LIN {X 0,Y 481.295,Z 335.256,A -85,B 0,C 180,E1 -6793.339,E2 -6793.339} C_VEL
LIN {X 0,Y 481.494,Z 329.441,A -85,B 0,C 180,E1 -6794.339,E2 -6794.339} C_VEL
LIN {X 0,Y 481.671,Z 324.523,A -85,B 0,C 180,E1 -6795.045,E2 -6795.045} C_VEL
LIN {X 0,Y 481.939,Z 317.288,A -85,B 0,C 180,E1 -6795.906,E2 -6795.906} C_VEL
LIN {X 0,Y 482.147,Z 309.914,A -85,B 0,C 180,E1 -6796.628,E2 -6796.628} C_VEL
LIN {X 0,Y 482.417,Z 301.623,A -85,B 0,C 180,E1 -6797.289,E2 -6797.289} C_VEL
LIN {X 0,Y 482.717,Z 290.959,A -85,B 0,C 180,E1 -6797.954,E2 -6797.954} C_VEL
LIN {X 0,Y 482.784,Z 280.373,A -85,B 0,C 180,E1 -6798.426,E2 -6798.426} C_VEL
LIN {X 0,Y 481.052,Z 270.815,A -85,B 0,C 180,E1 -6798.793,E2 -6798.793} C_VEL
LIN {X 0,Y 481.125,Z 264.772,A -85,B 0,C 180,E1 -6801.617,E2 -6801.617} C_VEL
LIN {X 0,Y 481.175,Z 257.779,A -85,B 0,C 180,E1 -6804.879,E2 -6804.879} C_VEL
LIN {X 0,Y 481.271,Z 252.542,A -85,B 0,C 180,E1 -6807.295,E2 -6807.295} C_VEL
LIN {X 0,Y 481.297,Z 246.12,A -85,B 0,C 180,E1 -6810.233,E2 -6810.233} C_VEL
LIN {X 0,Y 481.291,Z 239.614,A -85,B 0,C 180,E1 -6813.084,E2 -6813.084} C_VEL
LIN {X 0,Y 481.364,Z 233.224,A -85,B 0,C 180,E1 -6815.87,E2 -6815.87} C_VEL
LIN {X 0,Y 481.43,Z 228.524,A -85,B 0,C 180,E1 -6817.92,E2 -6817.92} C_VEL
LIN {X 0,Y 481.692,Z 228.485,A -85,B 0,C 180,E1 -6820.392,E2 -6820.392} C_VEL
LIN {X 0,Y 481.681,Z 228.487,A -85,B 0,C 180,E1 -6823.033,E2 -6823.033} C_VEL
LIN {X 0,Y 481.691,Z 228.486,A -85,B 0,C 180,E1 -6825.639,E2 -6825.639} C_VEL
LIN {X 0,Y 481.754,Z 228.48,A -85,B 0,C 180,E1 -6828.215,E2 -6828.215} C_VEL
LIN {X 0,Y 481.766,Z 228.477,A -85,B 0,C 180,E1 -6831.612,E2 -6831.612} C_VEL
LIN {X 0,Y 481.778,Z 228.474,A -85,B 0,C 180,E1 -6834.979,E2 -6834.979} C_VEL
LIN {X 0,Y 481.931,Z 228.456,A -85,B 0,C 180,E1 -6837.492,E2 -6837.492} C_VEL
LIN {X 0,Y 481.889,Z 228.46,A -85,B 0,C 180,E1 -6840.836,E2 -6840.836} C_VEL
LIN {X 0,Y 481.931,Z 228.458,A -85,B 0,C 180,E1 -6842.507,E2 -6842.507} C_VEL
LIN {X 0,Y 481.8,Z 228.472,A -85,B 0,C 180,E1 -6845.861,E2 -6845.861} C_VEL
LIN {X 0,Y 481.765,Z 228.477,A -85,B 0,C 180,E1 -6848.388,E2 -6848.388} C_VEL
LIN {X 0,Y 481.754,Z 228.477,A -85,B 0,C 180,E1 -6851.785,E2 -6851.785} C_VEL
LIN {X 0,Y 481.746,Z 228.478,A -85,B 0,C 180,E1 -6855.224,E2 -6855.224} C_VEL
LIN {X 0,Y 481.711,Z 228.481,A -85,B 0,C 180,E1 -6858.722,E2 -6858.722} C_VEL
LIN {X 0,Y 481.648,Z 228.491,A -85,B 0,C 180,E1 -6861.395,E2 -6861.395} C_VEL
LIN {X 0,Y 481.654,Z 228.489,A -85,B 0,C 180,E1 -6864.114,E2 -6864.114} C_VEL
LIN {X 0,Y 481.718,Z 228.48,A -85,B 0,C 180,E1 -6867.132,E2 -6867.132} C_VEL
LIN {X 0,Y 481.68,Z 228.486,A -85,B 0,C 180,E1 -6869.741,E2 -6869.741} C_VEL
LIN {X 0,Y 481.672,Z 228.486,A -85,B 0,C 180,E1 -6872.674,E2 -6872.674} C_VEL
LIN {X 0,Y 481.638,Z 228.492,A -85,B 0,C 180,E1 -6875.71,E2 -6875.71} C_VEL
LIN {X 0,Y 481.673,Z 228.486,A -85,B 0,C 180,E1 -6878.859,E2 -6878.859} C_VEL
LIN {X 0,Y 481.654,Z 228.49,A -85,B 0,C 180,E1 -6881.913,E2 -6881.913} C_VEL
LIN {X 0,Y 481.656,Z 228.49,A -85,B 0,C 180,E1 -6884.458,E2 -6884.458} C_VEL
LIN {X 0,Y 481.649,Z 228.491,A -85,B 0,C 180,E1 -6887.839,E2 -6887.839} C_VEL
LIN {X 0,Y 481.737,Z 228.644,A -85,B 0,C 180,E1 -6890.145,E2 -6890.145} C_VEL
LIN {X 0,Y 483.016,Z 236.207,A -85,B 0,C 180,E1 -6893.376,E2 -6893.376} C_VEL
LIN {X 0,Y 483.177,Z 240.208,A -85,B 0,C 180,E1 -6894.988,E2 -6894.988} C_VEL
LIN {X 0,Y 482.787,Z 248.025,A -85,B 0,C 180,E1 -6897.992,E2 -6897.992} C_VEL
LIN {X 0,Y 482.344,Z 256.819,A -85,B 0,C 180,E1 -6901.261,E2 -6901.261} C_VEL
LIN {X 0,Y 481.939,Z 266.411,A -85,B 0,C 180,E1 -6904.707,E2 -6904.707} C_VEL
LIN {X 0,Y 481.657,Z 274.969,A -85,B 0,C 180,E1 -6907.705,E2 -6907.705} C_VEL
LIN {X 0,Y 481.398,Z 284.073,A -85,B 0,C 180,E1 -6910.823,E2 -6910.823} C_VEL
LIN {X 0,Y 481.24,Z 293.194,A -85,B 0,C 180,E1 -6913.89,E2 -6913.89} C_VEL
LIN {X 0,Y 481.156,Z 296.798,A -85,B 0,C 180,E1 -6915.082,E2 -6915.082} C_VEL
LIN {X 0,Y 483.171,Z 311.724,A -85,B 0,C 180,E1 -6915.563,E2 -6915.563} C_VEL
LIN {X 0,Y 483.633,Z 316.455,A -85,B 0,C 180,E1 -6915.751,E2 -6915.751} C_VEL
LIN {X 0,Y 483.234,Z 328.917,A -85,B 0,C 180,E1 -6916.33,E2 -6916.33} C_VEL
LIN {X 0,Y 482.765,Z 340.987,A -85,B 0,C 180,E1 -6917.067,E2 -6917.067} C_VEL
LIN {X 0,Y 482.282,Z 352.197,A -85,B 0,C 180,E1 -6917.938,E2 -6917.938} C_VEL
LIN {X 0,Y 481.972,Z 361.764,A -85,B 0,C 180,E1 -6918.86,E2 -6918.86} C_VEL
LIN {X 0,Y 481.571,Z 370.781,A -85,B 0,C 180,E1 -6919.914,E2 -6919.914} C_VEL
LIN {X 0,Y 481.279,Z 379.611,A -85,B 0,C 180,E1 -6921.18,E2 -6921.18} C_VEL
LIN {X 0,Y 481.101,Z 386.663,A -85,B 0,C 180,E1 -6922.445,E2 -6922.445} C_VEL
LIN {X 0,Y 480.921,Z 392.764,A -85,B 0,C 180,E1 -6923.827,E2 -6923.827} C_VEL
LIN {X 0,Y 480.902,Z 396.727,A -85,B 0,C 180,E1 -6924.97,E2 -6924.97} C_VEL
LIN {X 0,Y 480.849,Z 399.059,A -85,B 0,C 180,E1 -6925.809,E2 -6925.809} C_VEL
LIN {X 0,Y 480.894,Z 400.958,A -85,B 0,C 180,E1 -6926.649,E2 -6926.649} C_VEL
LIN {X 0,Y 480.869,Z 402.379,A -85,B 0,C 180,E1 -6927.487,E2 -6927.487} C_VEL
LIN {X 0,Y 480.824,Z 403.378,A -85,B 0,C 180,E1 -6928.325,E2 -6928.325} C_VEL
LIN {X 0,Y 480.763,Z 403.977,A -85,B 0,C 180,E1 -6929.163,E2 -6929.163} C_VEL
LIN {X 0,Y 480.752,Z 404.178,A -85,B 0,C 180,E1 -6930,E2 -6930} C_VEL
LIN {X 0,Y 480.764,Z 403.933,A -85,B 0,C 180,E1 -6930.838,E2 -6930.838} C_VEL
LIN {X 0,Y 480.824,Z 403.286,A -85,B 0,C 180,E1 -6931.675,E2 -6931.675} C_VEL
LIN {X 0,Y 480.869,Z 402.238,A -85,B 0,C 180,E1 -6932.513,E2 -6932.513} C_VEL
LIN {X 0,Y 480.896,Z 400.77,A -85,B 0,C 180,E1 -6933.351,E2 -6933.351} C_VEL
LIN {X 0,Y 480.847,Z 397.7,A -85,B 0,C 180,E1 -6934.611,E2 -6934.611} C_VEL
LIN {X 0,Y 480.931,Z 393.56,A -85,B 0,C 180,E1 -6935.871,E2 -6935.871} C_VEL
LIN {X 0,Y 481.106,Z 387.196,A -85,B 0,C 180,E1 -6937.344,E2 -6937.344} C_VEL
LIN {X 0,Y 481.256,Z 380.258,A -85,B 0,C 180,E1 -6938.609,E2 -6938.609} C_VEL
LIN {X 0,Y 481.508,Z 371.668,A -85,B 0,C 180,E1 -6939.875,E2 -6939.875} C_VEL
LIN {X 0,Y 481.844,Z 362.847,A -85,B 0,C 180,E1 -6940.93,E2 -6940.93} C_VEL
LIN {X 0,Y 482.173,Z 352.482,A -85,B 0,C 180,E1 -6941.948,E2 -6941.948} C_VEL
LIN {X 0,Y 482.589,Z 341.383,A -85,B 0,C 180,E1 -6942.832,E2 -6942.832} C_VEL
LIN {X 0,Y 483.067,Z 329.672,A -85,B 0,C 180,E1 -6943.568,E2 -6943.568} C_VEL
LIN {X 0,Y 483.567,Z 316.581,A -85,B 0,C 180,E1 -6944.197,E2 -6944.197} C_VEL
LIN {X 0,Y 482.164,Z 303.16,A -85,B 0,C 180,E1 -6944.711,E2 -6944.711} C_VEL
LIN {X 0,Y 481.08,Z 295.296,A -85,B 0,C 180,E1 -6944.948,E2 -6944.948} C_VEL
LIN {X 0,Y 481.261,Z 284.885,A -85,B 0,C 180,E1 -6948.338,E2 -6948.338} C_VEL
LIN {X 0,Y 481.46,Z 275.744,A -85,B 0,C 180,E1 -6951.404,E2 -6951.404} C_VEL
LIN {X 0,Y 481.668,Z 266.683,A -85,B 0,C 180,E1 -6954.573,E2 -6954.573} C_VEL
LIN {X 0,Y 481.949,Z 259.603,A -85,B 0,C 180,E1 -6957.186,E2 -6957.186} C_VEL
LIN {X 0,Y 482.36,Z 252.034,A -85,B 0,C 180,E1 -6960.177,E2 -6960.177} C_VEL
LIN {X 0,Y 482.964,Z 245.384,A -85,B 0,C 180,E1 -6963.072,E2 -6963.072} C_VEL
LIN {X 0,Y 483.35,Z 240.369,A -85,B 0,C 180,E1 -6965.564,E2 -6965.564} C_VEL
LIN {X 0,Y 483.107,Z 236.847,A -85,B 0,C 180,E1 -6967.662,E2 -6967.662} C_VEL
LIN {X 0,Y 482.648,Z 233.878,A -85,B 0,C 180,E1 -6969.844,E2 -6969.844} C_VEL
LIN {X 0,Y 482.207,Z 231.543,A -85,B 0,C 180,E1 -6972.101,E2 -6972.101} C_VEL
LIN {X 0,Y 481.93,Z 229.935,A -85,B 0,C 180,E1 -6974.426,E2 -6974.426} C_VEL
LIN {X 0,Y 481.743,Z 229.06,A -85,B 0,C 180,E1 -6976.84,E2 -6976.84} C_VEL
LIN {X 0,Y 481.749,Z 228.914,A -85,B 0,C 180,E1 -6979.342,E2 -6979.342} C_VEL
LIN {X 0,Y 481.838,Z 229.553,A -85,B 0,C 180,E1 -6982.222,E2 -6982.222} C_VEL
LIN {X 0,Y 481.94,Z 230.974,A -85,B 0,C 180,E1 -6985.339,E2 -6985.339} C_VEL
LIN {X 0,Y 481.767,Z 232.856,A -85,B 0,C 180,E1 -6988.32,E2 -6988.32} C_VEL
LIN {X 0,Y 481.589,Z 234.985,A -85,B 0,C 180,E1 -6991.211,E2 -6991.211} C_VEL
LIN {X 0,Y 481.467,Z 237.269,A -85,B 0,C 180,E1 -6994.029,E2 -6994.029} C_VEL
LIN {X 0,Y 481.344,Z 239.756,A -85,B 0,C 180,E1 -6996.905,E2 -6996.905} C_VEL
LIN {X 0,Y 481.253,Z 242.102,A -85,B 0,C 180,E1 -6999.483,E2 -6999.483} C_VEL
LIN {X 0,Y 481.221,Z 244.619,A -85,B 0,C 180,E1 -7002.14,E2 -7002.14} C_VEL
LIN {X 0,Y 481.172,Z 247.192,A -85,B 0,C 180,E1 -7004.757,E2 -7004.757} C_VEL
LIN {X 0,Y 481.113,Z 248.8,A -85,B 0,C 180,E1 -7006.201,E2 -7006.201} C_VEL
LIN {X 0,Y 484.037,Z 261.107,A -85,B 0,C 180,E1 -7006.7,E2 -7006.7} C_VEL
LIN {X 0,Y 483.743,Z 273.649,A -85,B 0,C 180,E1 -7007.254,E2 -7007.254} C_VEL
LIN {X 0,Y 483.415,Z 285.282,A -85,B 0,C 180,E1 -7007.937,E2 -7007.937} C_VEL
LIN {X 0,Y 482.913,Z 296.516,A -85,B 0,C 180,E1 -7008.776,E2 -7008.776} C_VEL
LIN {X 0,Y 482.478,Z 306.707,A -85,B 0,C 180,E1 -7009.721,E2 -7009.721} C_VEL
LIN {X 0,Y 482.162,Z 315.925,A -85,B 0,C 180,E1 -7010.774,E2 -7010.774} C_VEL
LIN {X 0,Y 481.71,Z 324.854,A -85,B 0,C 180,E1 -7012.033,E2 -7012.033} C_VEL
LIN {X 0,Y 481.487,Z 332.04,A -85,B 0,C 180,E1 -7013.294,E2 -7013.294} C_VEL
LIN {X 0,Y 481.262,Z 337.788,A -85,B 0,C 180,E1 -7014.553,E2 -7014.553} C_VEL
LIN {X 0,Y 481.111,Z 342.296,A -85,B 0,C 180,E1 -7015.812,E2 -7015.812} C_VEL
LIN {X 0,Y 481.138,Z 344.659,A -85,B 0,C 180,E1 -7016.65,E2 -7016.65} C_VEL
LIN {X 0,Y 480.969,Z 346.601,A -85,B 0,C 180,E1 -7017.488,E2 -7017.488} C_VEL
LIN {X 0,Y 480.838,Z 348.127,A -85,B 0,C 180,E1 -7018.325,E2 -7018.325} C_VEL
LIN {X 0,Y 480.778,Z 349.206,A -85,B 0,C 180,E1 -7019.163,E2 -7019.163} C_VEL
LIN {X 0,Y 480.771,Z 350.142,A -85,B 0,C 180,E1 -7020.838,E2 -7020.838} C_VEL
LIN {X 0,Y 480.828,Z 350.027,A -85,B 0,C 180,E1 -7021.675,E2 -7021.675} C_VEL
LIN {X 0,Y 480.94,Z 349.479,A -85,B 0,C 180,E1 -7022.513,E2 -7022.513} C_VEL
LIN {X 0,Y 480.954,Z 348.529,A -85,B 0,C 180,E1 -7023.351,E2 -7023.351} C_VEL
LIN {X 0,Y 480.975,Z 347.183,A -85,B 0,C 180,E1 -7024.19,E2 -7024.19} C_VEL
LIN {X 0,Y 481.002,Z 344.348,A -85,B 0,C 180,E1 -7025.45,E2 -7025.45} C_VEL
LIN {X 0,Y 481.06,Z 340.212,A -85,B 0,C 180,E1 -7026.785,E2 -7026.785} C_VEL
LIN {X 0,Y 481.287,Z 335.46,A -85,B 0,C 180,E1 -7027.974,E2 -7027.974} C_VEL
LIN {X 0,Y 481.499,Z 329.153,A -85,B 0,C 180,E1 -7029.239,E2 -7029.239} C_VEL
LIN {X 0,Y 481.772,Z 321.248,A -85,B 0,C 180,E1 -7030.507,E2 -7030.507} C_VEL
LIN {X 0,Y 482.233,Z 311.394,A -85,B 0,C 180,E1 -7031.773,E2 -7031.773} C_VEL
LIN {X 0,Y 482.545,Z 302.284,A -85,B 0,C 180,E1 -7032.726,E2 -7032.726} C_VEL
LIN {X 0,Y 482.971,Z 290.987,A -85,B 0,C 180,E1 -7033.678,E2 -7033.678} C_VEL
LIN {X 0,Y 483.467,Z 279.995,A -85,B 0,C 180,E1 -7034.415,E2 -7034.415} C_VEL
LIN {X 0,Y 483.747,Z 267.916,A -85,B 0,C 180,E1 -7035.052,E2 -7035.052} C_VEL
LIN {X 0,Y 483.69,Z 259.543,A -85,B 0,C 180,E1 -7035.396,E2 -7035.396} C_VEL
LIN {X 0,Y 480.921,Z 246.835,A -85,B 0,C 180,E1 -7035.875,E2 -7035.875} C_VEL
LIN {X 0,Y 480.951,Z 243.537,A -85,B 0,C 180,E1 -7038.753,E2 -7038.753} C_VEL
LIN {X 0,Y 480.946,Z 240.512,A -85,B 0,C 180,E1 -7041.428,E2 -7041.428} C_VEL
LIN {X 0,Y 481.05,Z 236.454,A -85,B 0,C 180,E1 -7045.067,E2 -7045.067} C_VEL
LIN {X 0,Y 481.082,Z 233.378,A -85,B 0,C 180,E1 -7047.871,E2 -7047.871} C_VEL
LIN {X 0,Y 481.1,Z 230.253,A -85,B 0,C 180,E1 -7050.75,E2 -7050.75} C_VEL
LIN {X 0,Y 481.116,Z 228.819,A -85,B 0,C 180,E1 -7052.086,E2 -7052.086} C_VEL
LIN {X 0,Y 481.303,Z 228.535,A -85,B 0,C 180,E1 -7053.703,E2 -7053.703} C_VEL
LIN {X 0,Y 481.586,Z 228.499,A -85,B 0,C 180,E1 -7056.616,E2 -7056.616} C_VEL
LIN {X 0,Y 481.66,Z 228.487,A -85,B 0,C 180,E1 -7059.345,E2 -7059.345} C_VEL
LIN {X 0,Y 481.648,Z 228.49,A -85,B 0,C 180,E1 -7062.161,E2 -7062.161} C_VEL
LIN {X 0,Y 481.658,Z 228.489,A -85,B 0,C 180,E1 -7065.542,E2 -7065.542} C_VEL
LIN {X 0,Y 481.632,Z 228.493,A -85,B 0,C 180,E1 -7068.955,E2 -7068.955} C_VEL
LIN {X 0,Y 481.63,Z 228.488,A -85,B 0,C 180,E1 -7071.997,E2 -7071.997} C_VEL
LIN {X 0,Y 481.681,Z 228.482,A -85,B 0,C 180,E1 -7075.317,E2 -7075.317} C_VEL
LIN {X 0,Y 481.647,Z 228.491,A -85,B 0,C 180,E1 -7078.311,E2 -7078.311} C_VEL
LIN {X 0,Y 481.679,Z 228.483,A -85,B 0,C 180,E1 -7081.217,E2 -7081.217} C_VEL
LIN {X 0,Y 481.68,Z 228.484,A -85,B 0,C 180,E1 -7082.587,E2 -7082.587} C_VEL
LIN {X 0,Y 481.036,Z 228.564,A -85,B 0,C 180,E1 -7083.285,E2 -7083.285} C_VEL
LIN {X 0,Y 478.166,Z 228.923,A -85,B 0,C 180,E1 -7084.417,E2 -7084.417} C_VEL
LIN {X 0,Y 475.728,Z 229.227,A -85,B 0,C 180,E1 -7085.33,E2 -7085.33} C_VEL
LIN {X 0,Y 474.689,Z 229.358,A -85,B 0,C 180,E1 -7086.036,E2 -7086.036} C_VEL
LIN {X 0,Y 474.609,Z 229.364,A -85,B 0,C 180,E1 -7086.275,E2 -7086.275} C_VEL
LIN {X 0,Y 474.675,Z 229.358,A -85,B 0,C 180,E1 -7089.185,E2 -7089.185} C_VEL
LIN {X 0,Y 474.65,Z 229.36,A -85,B 0,C 180,E1 -7091.884,E2 -7091.884} C_VEL
LIN {X 0,Y 474.703,Z 229.355,A -85,B 0,C 180,E1 -7094.544,E2 -7094.544} C_VEL
LIN {X 0,Y 474.708,Z 229.353,A -85,B 0,C 180,E1 -7098.037,E2 -7098.037} C_VEL
LIN {X 0,Y 474.7,Z 229.352,A -85,B 0,C 180,E1 -7101.486,E2 -7101.486} C_VEL
LIN {X 0,Y 474.73,Z 229.354,A -85,B 0,C 180,E1 -7104.052,E2 -7104.052} C_VEL
LIN {X 0,Y 474.874,Z 229.332,A -85,B 0,C 180,E1 -7107.455,E2 -7107.455} C_VEL
LIN {X 0,Y 474.887,Z 229.331,A -85,B 0,C 180,E1 -7110,E2 -7110} C_VEL
LIN {X 0,Y 474.889,Z 229.328,A -85,B 0,C 180,E1 -7112.545,E2 -7112.545} C_VEL
LIN {X 0,Y 474.461,Z 229.391,A -85,B 0,C 180,E1 -7115.738,E2 -7115.738} C_VEL
LIN {X 0,Y 474.408,Z 229.618,A -85,B 0,C 180,E1 -7115.952,E2 -7115.952} C_VEL
LIN {X 0,Y 474.316,Z 235.276,A -85,B 0,C 180,E1 -7118.521,E2 -7118.521} C_VEL
LIN {X 0,Y 474.336,Z 242.968,A -85,B 0,C 180,E1 -7122.069,E2 -7122.069} C_VEL
LIN {X 0,Y 474.215,Z 250.471,A -85,B 0,C 180,E1 -7125.565,E2 -7125.565} C_VEL
LIN {X 0,Y 474.13,Z 256.598,A -85,B 0,C 180,E1 -7128.437,E2 -7128.437} C_VEL
LIN {X 0,Y 474.012,Z 263.644,A -85,B 0,C 180,E1 -7131.757,E2 -7131.757} C_VEL
LIN {X 0,Y 474.035,Z 270.842,A -85,B 0,C 180,E1 -7135.149,E2 -7135.149} C_VEL
LIN {X 0,Y 475.886,Z 281.886,A -85,B 0,C 180,E1 -7135.561,E2 -7135.561} C_VEL
LIN {X 0,Y 475.639,Z 293.378,A -85,B 0,C 180,E1 -7136.119,E2 -7136.119} C_VEL
LIN {X 0,Y 475.361,Z 302.095,A -85,B 0,C 180,E1 -7136.685,E2 -7136.685} C_VEL
LIN {X 0,Y 475.169,Z 309.613,A -85,B 0,C 180,E1 -7137.291,E2 -7137.291} C_VEL
LIN {X 0,Y 474.932,Z 317.222,A -85,B 0,C 180,E1 -7138.038,E2 -7138.038} C_VEL
LIN {X 0,Y 474.695,Z 323.363,A -85,B 0,C 180,E1 -7138.762,E2 -7138.762} C_VEL
LIN {X 0,Y 474.499,Z 328.691,A -85,B 0,C 180,E1 -7139.504,E2 -7139.504} C_VEL
LIN {X 0,Y 474.263,Z 334.555,A -85,B 0,C 180,E1 -7140.491,E2 -7140.491} C_VEL
LIN {X 0,Y 474.117,Z 339.399,A -85,B 0,C 180,E1 -7141.502,E2 -7141.502} C_VEL
LIN {X 0,Y 473.929,Z 344.143,A -85,B 0,C 180,E1 -7142.77,E2 -7142.77} C_VEL
LIN {X 0,Y 473.879,Z 347.053,A -85,B 0,C 180,E1 -7143.847,E2 -7143.847} C_VEL
LIN {X 0,Y 473.719,Z 349.579,A -85,B 0,C 180,E1 -7145.352,E2 -7145.352} C_VEL
LIN {X 0,Y 473.688,Z 350.576,A -85,B 0,C 180,E1 -7146.756,E2 -7146.756} C_VEL
LIN {X 0,Y 473.672,Z 350.258,A -85,B 0,C 180,E1 -7148.151,E2 -7148.151} C_VEL
LIN {X 0,Y 473.795,Z 348.314,A -85,B 0,C 180,E1 -7149.631,E2 -7149.631} C_VEL
LIN {X 0,Y 473.903,Z 345.887,A -85,B 0,C 180,E1 -7150.732,E2 -7150.732} C_VEL
LIN {X 0,Y 474.004,Z 342.445,A -85,B 0,C 180,E1 -7151.852,E2 -7151.852} C_VEL
LIN {X 0,Y 474.228,Z 336.841,A -85,B 0,C 180,E1 -7153.206,E2 -7153.206} C_VEL
LIN {X 0,Y 474.472,Z 330.093,A -85,B 0,C 180,E1 -7154.407,E2 -7154.407} C_VEL
LIN {X 0,Y 474.705,Z 323.97,A -85,B 0,C 180,E1 -7155.287,E2 -7155.287} C_VEL
LIN {X 0,Y 474.967,Z 316.576,A -85,B 0,C 180,E1 -7156.159,E2 -7156.159} C_VEL
LIN {X 0,Y 475.319,Z 307.718,A -85,B 0,C 180,E1 -7157.004,E2 -7157.004} C_VEL
LIN {X 0,Y 475.552,Z 297.935,A -85,B 0,C 180,E1 -7157.723,E2 -7157.723} C_VEL
LIN {X 0,Y 475.811,Z 288.494,A -85,B 0,C 180,E1 -7158.255,E2 -7158.255} C_VEL
LIN {X 0,Y 475.789,Z 280.908,A -85,B 0,C 180,E1 -7158.591,E2 -7158.591} C_VEL
LIN {X 0,Y 474.005,Z 271.202,A -85,B 0,C 180,E1 -7158.96,E2 -7158.96} C_VEL
LIN {X 0,Y 474.078,Z 265.171,A -85,B 0,C 180,E1 -7161.786,E2 -7161.786} C_VEL
LIN {X 0,Y 474.14,Z 257.884,A -85,B 0,C 180,E1 -7165.203,E2 -7165.203} C_VEL
LIN {X 0,Y 474.209,Z 252.36,A -85,B 0,C 180,E1 -7167.755,E2 -7167.755} C_VEL
LIN {X 0,Y 474.264,Z 245.792,A -85,B 0,C 180,E1 -7170.724,E2 -7170.724} C_VEL
LIN {X 0,Y 474.267,Z 238.22,A -85,B 0,C 180,E1 -7174.078,E2 -7174.078} C_VEL
LIN {X 0,Y 474.304,Z 232.086,A -85,B 0,C 180,E1 -7176.735,E2 -7176.735} C_VEL
LIN {X 0,Y 474.397,Z 229.401,A -85,B 0,C 180,E1 -7177.919,E2 -7177.919} C_VEL
LIN {X 0,Y 474.631,Z 229.366,A -85,B 0,C 180,E1 -7180.088,E2 -7180.088} C_VEL
LIN {X 0,Y 474.641,Z 229.364,A -85,B 0,C 180,E1 -7182.774,E2 -7182.774} C_VEL
LIN {X 0,Y 474.65,Z 229.362,A -85,B 0,C 180,E1 -7185.421,E2 -7185.421} C_VEL
LIN {X 0,Y 474.708,Z 229.357,A -85,B 0,C 180,E1 -7188.038,E2 -7188.038} C_VEL
LIN {X 0,Y 474.731,Z 229.352,A -85,B 0,C 180,E1 -7191.486,E2 -7191.486} C_VEL
LIN {X 0,Y 474.748,Z 229.35,A -85,B 0,C 180,E1 -7194.904,E2 -7194.904} C_VEL
LIN {X 0,Y 474.897,Z 229.332,A -85,B 0,C 180,E1 -7197.455,E2 -7197.455} C_VEL
LIN {X 0,Y 474.915,Z 229.33,A -85,B 0,C 180,E1 -7200,E2 -7200} C_VEL
LIN {X 0,Y 474.897,Z 229.334,A -85,B 0,C 180,E1 -7202.545,E2 -7202.545} C_VEL
LIN {X 0,Y 474.761,Z 229.349,A -85,B 0,C 180,E1 -7205.948,E2 -7205.948} C_VEL
LIN {X 0,Y 474.73,Z 229.353,A -85,B 0,C 180,E1 -7208.513,E2 -7208.513} C_VEL
LIN {X 0,Y 474.708,Z 229.356,A -85,B 0,C 180,E1 -7211.962,E2 -7211.962} C_VEL
LIN {X 0,Y 474.703,Z 229.357,A -85,B 0,C 180,E1 -7215.456,E2 -7215.456} C_VEL
LIN {X 0,Y 474.665,Z 229.36,A -85,B 0,C 180,E1 -7219.01,E2 -7219.01} C_VEL
LIN {X 0,Y 474.591,Z 229.37,A -85,B 0,C 180,E1 -7221.729,E2 -7221.729} C_VEL
LIN {X 0,Y 474.632,Z 229.363,A -85,B 0,C 180,E1 -7224.494,E2 -7224.494} C_VEL
LIN {X 0,Y 474.675,Z 229.358,A -85,B 0,C 180,E1 -7227.332,E2 -7227.332} C_VEL
LIN {X 0,Y 474.606,Z 229.367,A -85,B 0,C 180,E1 -7230.23,E2 -7230.23} C_VEL
LIN {X 0,Y 474.627,Z 229.365,A -85,B 0,C 180,E1 -7233.221,E2 -7233.221} C_VEL
LIN {X 0,Y 474.591,Z 229.368,A -85,B 0,C 180,E1 -7236.323,E2 -7236.323} C_VEL
LIN {X 0,Y 474.63,Z 229.364,A -85,B 0,C 180,E1 -7239.648,E2 -7239.648} C_VEL
LIN {X 0,Y 474.616,Z 229.368,A -85,B 0,C 180,E1 -7242.934,E2 -7242.934} C_VEL
LIN {X 0,Y 474.608,Z 229.368,A -85,B 0,C 180,E1 -7245.895,E2 -7245.895} C_VEL
LIN {X 0,Y 474.629,Z 229.365,A -85,B 0,C 180,E1 -7249.041,E2 -7249.041} C_VEL
LIN {X 0,Y 474.665,Z 229.461,A -85,B 0,C 180,E1 -7249.875,E2 -7249.875} C_VEL
LIN {X 0,Y 475.873,Z 236.391,A -85,B 0,C 180,E1 -7252.893,E2 -7252.893} C_VEL
LIN {X 0,Y 476.198,Z 241.158,A -85,B 0,C 180,E1 -7254.859,E2 -7254.859} C_VEL
LIN {X 0,Y 475.794,Z 248.869,A -85,B 0,C 180,E1 -7257.876,E2 -7257.876} C_VEL
LIN {X 0,Y 475.373,Z 256.603,A -85,B 0,C 180,E1 -7260.799,E2 -7260.799} C_VEL
LIN {X 0,Y 474.982,Z 265.641,A -85,B 0,C 180,E1 -7264.12,E2 -7264.12} C_VEL
LIN {X 0,Y 474.622,Z 274.707,A -85,B 0,C 180,E1 -7267.356,E2 -7267.356} C_VEL
LIN {X 0,Y 474.342,Z 283.791,A -85,B 0,C 180,E1 -7270.527,E2 -7270.527} C_VEL
LIN {X 0,Y 474.129,Z 294.299,A -85,B 0,C 180,E1 -7274.128,E2 -7274.128} C_VEL
LIN {X 0,Y 474.095,Z 296.6,A -85,B 0,C 180,E1 -7274.882,E2 -7274.882} C_VEL
LIN {X 0,Y 475.967,Z 310.299,A -85,B 0,C 180,E1 -7275.312,E2 -7275.312} C_VEL
LIN {X 0,Y 476.688,Z 317.105,A -85,B 0,C 180,E1 -7275.594,E2 -7275.594} C_VEL
LIN {X 0,Y 476.225,Z 330.263,A -85,B 0,C 180,E1 -7276.233,E2 -7276.233} C_VEL
LIN {X 0,Y 475.738,Z 341.948,A -85,B 0,C 180,E1 -7276.98,E2 -7276.98} C_VEL
LIN {X 0,Y 475.237,Z 352.96,A -85,B 0,C 180,E1 -7277.876,E2 -7277.876} C_VEL
LIN {X 0,Y 474.866,Z 363.214,A -85,B 0,C 180,E1 -7278.907,E2 -7278.907} C_VEL
LIN {X 0,Y 474.471,Z 371.932,A -85,B 0,C 180,E1 -7279.977,E2 -7279.977} C_VEL
LIN {X 0,Y 474.178,Z 380.414,A -85,B 0,C 180,E1 -7281.262,E2 -7281.262} C_VEL
LIN {X 0,Y 474.013,Z 387.242,A -85,B 0,C 180,E1 -7282.546,E2 -7282.546} C_VEL
LIN {X 0,Y 473.836,Z 393.505,A -85,B 0,C 180,E1 -7284.041,E2 -7284.041} C_VEL
LIN {X 0,Y 473.764,Z 397.562,A -85,B 0,C 180,E1 -7285.32,E2 -7285.32} C_VEL
LIN {X 0,Y 473.82,Z 400.554,A -85,B 0,C 180,E1 -7286.599,E2 -7286.599} C_VEL
LIN {X 0,Y 473.783,Z 401.98,A -85,B 0,C 180,E1 -7287.45,E2 -7287.45} C_VEL
LIN {X 0,Y 473.758,Z 402.981,A -85,B 0,C 180,E1 -7288.3,E2 -7288.3} C_VEL
LIN {X 0,Y 473.692,Z 403.58,A -85,B 0,C 180,E1 -7289.15,E2 -7289.15} C_VEL
LIN {X 0,Y 473.678,Z 403.781,A -85,B 0,C 180,E1 -7290,E2 -7290} C_VEL
LIN {X 0,Y 473.692,Z 403.535,A -85,B 0,C 180,E1 -7290.85,E2 -7290.85} C_VEL
LIN {X 0,Y 473.758,Z 402.883,A -85,B 0,C 180,E1 -7291.7,E2 -7291.7} C_VEL
LIN {X 0,Y 473.783,Z 401.827,A -85,B 0,C 180,E1 -7292.551,E2 -7292.551} C_VEL
LIN {X 0,Y 473.822,Z 400.353,A -85,B 0,C 180,E1 -7293.402,E2 -7293.402} C_VEL
LIN {X 0,Y 473.77,Z 397.27,A -85,B 0,C 180,E1 -7294.68,E2 -7294.68} C_VEL
LIN {X 0,Y 473.824,Z 392.416,A -85,B 0,C 180,E1 -7296.141,E2 -7296.141} C_VEL
LIN {X 0,Y 474.014,Z 386.74,A -85,B 0,C 180,E1 -7297.454,E2 -7297.454} C_VEL
LIN {X 0,Y 474.166,Z 379.794,A -85,B 0,C 180,E1 -7298.739,E2 -7298.739} C_VEL
LIN {X 0,Y 474.446,Z 371.188,A -85,B 0,C 180,E1 -7300.024,E2 -7300.024} C_VEL
LIN {X 0,Y 474.828,Z 362.369,A -85,B 0,C 180,E1 -7301.094,E2 -7301.094} C_VEL
LIN {X 0,Y 475.18,Z 352.261,A -85,B 0,C 180,E1 -7302.105,E2 -7302.105} C_VEL
LIN {X 0,Y 475.642,Z 340.961,A -85,B 0,C 180,E1 -7303.023,E2 -7303.023} C_VEL
LIN {X 0,Y 476.16,Z 329.303,A -85,B 0,C 180,E1 -7303.769,E2 -7303.769} C_VEL
LIN {X 0,Y 476.673,Z 316.331,A -85,B 0,C 180,E1 -7304.407,E2 -7304.407} C_VEL
LIN {X 0,Y 475.204,Z 303.316,A -85,B 0,C 180,E1 -7304.931,E2 -7304.931} C_VEL
LIN {X 0,Y 474,Z 294.784,A -85,B 0,C 180,E1 -7305.204,E2 -7305.204} C_VEL
LIN {X 0,Y 474.184,Z 285.008,A -85,B 0,C 180,E1 -7308.457,E2 -7308.457} C_VEL
LIN {X 0,Y 474.438,Z 275.456,A -85,B 0,C 180,E1 -7311.736,E2 -7311.736} C_VEL
LIN {X 0,Y 474.661,Z 266.492,A -85,B 0,C 180,E1 -7314.96,E2 -7314.96} C_VEL
LIN {X 0,Y 474.998,Z 259.102,A -85,B 0,C 180,E1 -7317.779,E2 -7317.779} C_VEL
LIN {X 0,Y 475.539,Z 250.953,A -85,B 0,C 180,E1 -7321.149,E2 -7321.149} C_VEL
LIN {X 0,Y 476.199,Z 244.574,A -85,B 0,C 180,E1 -7324.113,E2 -7324.113} C_VEL
LIN {X 0,Y 476.345,Z 240.753,A -85,B 0,C 180,E1 -7326.169,E2 -7326.169} C_VEL
LIN {X 0,Y 476.008,Z 237.146,A -85,B 0,C 180,E1 -7328.508,E2 -7328.508} C_VEL
LIN {X 0,Y 475.481,Z 234.101,A -85,B 0,C 180,E1 -7331.077,E2 -7331.077} C_VEL
LIN {X 0,Y 475.034,Z 231.717,A -85,B 0,C 180,E1 -7334.056,E2 -7334.056} C_VEL
LIN {X 0,Y 474.807,Z 230.54,A -85,B 0,C 180,E1 -7337.087,E2 -7337.087} C_VEL
LIN {X 0,Y 474.809,Z 230.383,A -85,B 0,C 180,E1 -7339.362,E2 -7339.362} C_VEL
LIN {X 0,Y 474.841,Z 230.755,A -85,B 0,C 180,E1 -7341.67,E2 -7341.67} C_VEL
LIN {X 0,Y 474.956,Z 231.92,A -85,B 0,C 180,E1 -7344.754,E2 -7344.754} C_VEL
LIN {X 0,Y 474.833,Z 233.486,A -85,B 0,C 180,E1 -7347.529,E2 -7347.529} C_VEL
LIN {X 0,Y 474.674,Z 234.984,A -85,B 0,C 180,E1 -7349.775,E2 -7349.775} C_VEL
LIN {X 0,Y 474.517,Z 237.197,A -85,B 0,C 180,E1 -7352.705,E2 -7352.705} C_VEL
LIN {X 0,Y 474.363,Z 239.473,A -85,B 0,C 180,E1 -7355.491,E2 -7355.491} C_VEL
LIN {X 0,Y 474.234,Z 241.881,A -85,B 0,C 180,E1 -7358.254,E2 -7358.254} C_VEL
LIN {X 0,Y 474.185,Z 245.194,A -85,B 0,C 180,E1 -7361.866,E2 -7361.866} C_VEL
LIN {X 0,Y 474.14,Z 247.761,A -85,B 0,C 180,E1 -7364.526,E2 -7364.526} C_VEL
LIN {X 0,Y 474.052,Z 249.317,A -85,B 0,C 180,E1 -7365.95,E2 -7365.95} C_VEL
LIN {X 0,Y 477.224,Z 262.361,A -85,B 0,C 180,E1 -7366.505,E2 -7366.505} C_VEL
LIN {X 0,Y 476.875,Z 274.641,A -85,B 0,C 180,E1 -7367.066,E2 -7367.066} C_VEL
LIN {X 0,Y 476.518,Z 286.091,A -85,B 0,C 180,E1 -7367.76,E2 -7367.76} C_VEL
LIN {X 0,Y 475.995,Z 297.222,A -85,B 0,C 180,E1 -7368.61,E2 -7368.61} C_VEL
LIN {X 0,Y 475.538,Z 307.345,A -85,B 0,C 180,E1 -7369.57,E2 -7369.57} C_VEL
LIN {X 0,Y 475.189,Z 316.515,A -85,B 0,C 180,E1 -7370.637,E2 -7370.637} C_VEL
LIN {X 0,Y 474.708,Z 325.404,A -85,B 0,C 180,E1 -7371.915,E2 -7371.915} C_VEL
LIN {X 0,Y 474.46,Z 332.559,A -85,B 0,C 180,E1 -7373.194,E2 -7373.194} C_VEL
LIN {X 0,Y 474.224,Z 338.281,A -85,B 0,C 180,E1 -7374.472,E2 -7374.472} C_VEL
LIN {X 0,Y 474.063,Z 342.774,A -85,B 0,C 180,E1 -7375.749,E2 -7375.749} C_VEL
LIN {X 0,Y 474.088,Z 345.126,A -85,B 0,C 180,E1 -7376.601,E2 -7376.601} C_VEL
LIN {X 0,Y 473.913,Z 347.058,A -85,B 0,C 180,E1 -7377.45,E2 -7377.45} C_VEL
LIN {X 0,Y 473.773,Z 348.574,A -85,B 0,C 180,E1 -7378.3,E2 -7378.3} C_VEL
LIN {X 0,Y 473.706,Z 349.636,A -85,B 0,C 180,E1 -7379.15,E2 -7379.15} C_VEL
LIN {X 0,Y 473.699,Z 350.548,A -85,B 0,C 180,E1 -7380.85,E2 -7380.85} C_VEL
LIN {X 0,Y 473.763,Z 350.419,A -85,B 0,C 180,E1 -7381.7,E2 -7381.7} C_VEL
LIN {X 0,Y 473.863,Z 349.851,A -85,B 0,C 180,E1 -7382.55,E2 -7382.55} C_VEL
LIN {X 0,Y 473.881,Z 348.886,A -85,B 0,C 180,E1 -7383.401,E2 -7383.401} C_VEL
LIN {X 0,Y 473.897,Z 347.526,A -85,B 0,C 180,E1 -7384.253,E2 -7384.253} C_VEL
LIN {X 0,Y 473.95,Z 344.659,A -85,B 0,C 180,E1 -7385.531,E2 -7385.531} C_VEL
LIN {X 0,Y 474.009,Z 340.754,A -85,B 0,C 180,E1 -7386.812,E2 -7386.812} C_VEL
LIN {X 0,Y 474.233,Z 335.699,A -85,B 0,C 180,E1 -7388.094,E2 -7388.094} C_VEL
LIN {X 0,Y 474.478,Z 329.343,A -85,B 0,C 180,E1 -7389.377,E2 -7389.377} C_VEL
LIN {X 0,Y 474.785,Z 321.372,A -85,B 0,C 180,E1 -7390.663,E2 -7390.663} C_VEL
LIN {X 0,Y 475.274,Z 311.462,A -85,B 0,C 180,E1 -7391.948,E2 -7391.948} C_VEL
LIN {X 0,Y 475.58,Z 302.268,A -85,B 0,C 180,E1 -7392.916,E2 -7392.916} C_VEL
LIN {X 0,Y 476.066,Z 290.878,A -85,B 0,C 180,E1 -7393.88,E2 -7393.88} C_VEL
LIN {X 0,Y 476.57,Z 279.793,A -85,B 0,C 180,E1 -7394.628,E2 -7394.628} C_VEL
LIN {X 0,Y 476.884,Z 267.517,A -85,B 0,C 180,E1 -7395.274,E2 -7395.274} C_VEL
LIN {X 0,Y 476.825,Z 260.682,A -85,B 0,C 180,E1 -7395.561,E2 -7395.561} C_VEL
LIN {X 0,Y 473.846,Z 247.161,A -85,B 0,C 180,E1 -7396.084,E2 -7396.084} C_VEL
LIN {X 0,Y 473.86,Z 243.782,A -85,B 0,C 180,E1 -7399.044,E2 -7399.044} C_VEL
LIN {X 0,Y 473.872,Z 240.731,A -85,B 0,C 180,E1 -7401.764,E2 -7401.764} C_VEL
LIN {X 0,Y 473.973,Z 236.87,A -85,B 0,C 180,E1 -7405.243,E2 -7405.243} C_VEL
LIN {X 0,Y 474.001,Z 233.523,A -85,B 0,C 180,E1 -7408.325,E2 -7408.325} C_VEL
LIN {X 0,Y 474.021,Z 230.358,A -85,B 0,C 180,E1 -7411.26,E2 -7411.26} C_VEL
LIN {X 0,Y 474.088,Z 229.434,A -85,B 0,C 180,E1 -7412.329,E2 -7412.329} C_VEL
LIN {X 0,Y 474.471,Z 229.387,A -85,B 0,C 180,E1 -7415.444,E2 -7415.444} C_VEL
LIN {X 0,Y 474.605,Z 229.368,A -85,B 0,C 180,E1 -7418.458,E2 -7418.458} C_VEL
LIN {X 0,Y 474.619,Z 229.366,A -85,B 0,C 180,E1 -7421.786,E2 -7421.786} C_VEL
LIN {X 0,Y 474.62,Z 229.367,A -85,B 0,C 180,E1 -7425.298,E2 -7425.298} C_VEL
LIN {X 0,Y 474.604,Z 229.364,A -85,B 0,C 180,E1 -7428.212,E2 -7428.212} C_VEL
LIN {X 0,Y 474.62,Z 229.363,A -85,B 0,C 180,E1 -7430.451,E2 -7430.451} C_VEL
LIN {X 0,Y 474.572,Z 229.366,A -85,B 0,C 180,E1 -7433.675,E2 -7433.675} C_VEL
LIN {X 0,Y 474.618,Z 229.366,A -85,B 0,C 180,E1 -7436.778,E2 -7436.778} C_VEL
LIN {X 0,Y 474.605,Z 229.365,A -85,B 0,C 180,E1 -7439.769,E2 -7439.769} C_VEL
LIN {X 0,Y 474.641,Z 229.361,A -85,B 0,C 180,E1 -7442.676,E2 -7442.676} C_VEL
LIN {X 0,Y 474.641,Z 229.362,A -85,B 0,C 180,E1 -7445.506,E2 -7445.506} C_VEL
LIN {X 0,Y 474.609,Z 229.364,A -85,B 0,C 180,E1 -7446.275,E2 -7446.275} C_VEL
LIN {X 0,Y 473.963,Z 229.447,A -85,B 0,C 180,E1 -7446.984,E2 -7446.984} C_VEL
LIN {X 0,Y 471.14,Z 229.803,A -85,B 0,C 180,E1 -7448.135,E2 -7448.135} C_VEL
LIN {X 0,Y 468.74,Z 230.101,A -85,B 0,C 180,E1 -7449.063,E2 -7449.063} C_VEL
LIN {X 0,Y 467.702,Z 230.228,A -85,B 0,C 180,E1 -7449.78,E2 -7449.78} C_VEL
LIN {X 0,Y 467.615,Z 230.237,A -85,B 0,C 180,E1 -7450.023,E2 -7450.023} C_VEL
LIN {X 0,Y 467.601,Z 230.238,A -85,B 0,C 180,E1 -7452.506,E2 -7452.506} C_VEL
LIN {X 0,Y 467.607,Z 230.238,A -85,B 0,C 180,E1 -7455.196,E2 -7455.196} C_VEL
LIN {X 0,Y 467.66,Z 230.23,A -85,B 0,C 180,E1 -7457.854,E2 -7457.854} C_VEL
LIN {X 0,Y 467.66,Z 230.229,A -85,B 0,C 180,E1 -7461.357,E2 -7461.357} C_VEL
LIN {X 0,Y 467.696,Z 230.229,A -85,B 0,C 180,E1 -7463.962,E2 -7463.962} C_VEL
LIN {X 0,Y 467.814,Z 230.211,A -85,B 0,C 180,E1 -7467.417,E2 -7467.417} C_VEL
LIN {X 0,Y 467.856,Z 230.207,A -85,B 0,C 180,E1 -7470,E2 -7470} C_VEL
LIN {X 0,Y 467.854,Z 230.204,A -85,B 0,C 180,E1 -7472.583,E2 -7472.583} C_VEL
LIN {X 0,Y 467.406,Z 230.269,A -85,B 0,C 180,E1 -7475.825,E2 -7475.825} C_VEL
LIN {X 0,Y 467.252,Z 236.356,A -85,B 0,C 180,E1 -7478.651,E2 -7478.651} C_VEL
LIN {X 0,Y 467.261,Z 243.956,A -85,B 0,C 180,E1 -7482.156,E2 -7482.156} C_VEL
LIN {X 0,Y 467.152,Z 251.56,A -85,B 0,C 180,E1 -7485.712,E2 -7485.712} C_VEL
LIN {X 0,Y 467.067,Z 257.611,A -85,B 0,C 180,E1 -7488.563,E2 -7488.563} C_VEL
LIN {X 0,Y 466.922,Z 265.106,A -85,B 0,C 180,E1 -7492.104,E2 -7492.104} C_VEL
LIN {X 0,Y 466.989,Z 271.27,A -85,B 0,C 180,E1 -7494.984,E2 -7494.984} C_VEL
LIN {X 0,Y 468.732,Z 281.223,A -85,B 0,C 180,E1 -7495.352,E2 -7495.352} C_VEL
LIN {X 0,Y 468.825,Z 287.104,A -85,B 0,C 180,E1 -7495.614,E2 -7495.614} C_VEL
LIN {X 0,Y 468.604,Z 296.086,A -85,B 0,C 180,E1 -7496.105,E2 -7496.105} C_VEL
LIN {X 0,Y 468.374,Z 303.616,A -85,B 0,C 180,E1 -7496.624,E2 -7496.624} C_VEL
LIN {X 0,Y 468.101,Z 312.096,A -85,B 0,C 180,E1 -7497.345,E2 -7497.345} C_VEL
LIN {X 0,Y 467.789,Z 320.648,A -85,B 0,C 180,E1 -7498.246,E2 -7498.246} C_VEL
LIN {X 0,Y 467.496,Z 328.555,A -85,B 0,C 180,E1 -7499.316,E2 -7499.316} C_VEL
LIN {X 0,Y 467.268,Z 334.184,A -85,B 0,C 180,E1 -7500.256,E2 -7500.256} C_VEL
LIN {X 0,Y 467.07,Z 339.392,A -85,B 0,C 180,E1 -7501.334,E2 -7501.334} C_VEL
LIN {X 0,Y 466.913,Z 342.651,A -85,B 0,C 180,E1 -7502.163,E2 -7502.163} C_VEL
LIN {X 0,Y 466.808,Z 346.227,A -85,B 0,C 180,E1 -7503.334,E2 -7503.334} C_VEL
LIN {X 0,Y 466.775,Z 348.008,A -85,B 0,C 180,E1 -7504.095,E2 -7504.095} C_VEL
LIN {X 0,Y 466.698,Z 349.474,A -85,B 0,C 180,E1 -7504.907,E2 -7504.907} C_VEL
LIN {X 0,Y 466.634,Z 350.64,A -85,B 0,C 180,E1 -7505.971,E2 -7505.971} C_VEL
LIN {X 0,Y 466.602,Z 351.046,A -85,B 0,C 180,E1 -7507.048,E2 -7507.048} C_VEL
LIN {X 0,Y 466.615,Z 350.361,A -85,B 0,C 180,E1 -7508.444,E2 -7508.444} C_VEL
LIN {X 0,Y 466.694,Z 349.48,A -85,B 0,C 180,E1 -7509.234,E2 -7509.234} C_VEL
LIN {X 0,Y 466.799,Z 347.417,A -85,B 0,C 180,E1 -7510.346,E2 -7510.346} C_VEL
LIN {X 0,Y 466.909,Z 344.366,A -85,B 0,C 180,E1 -7511.475,E2 -7511.475} C_VEL
LIN {X 0,Y 467.109,Z 338.968,A -85,B 0,C 180,E1 -7512.908,E2 -7512.908} C_VEL
LIN {X 0,Y 467.326,Z 333.219,A -85,B 0,C 180,E1 -7514.071,E2 -7514.071} C_VEL
LIN {X 0,Y 467.659,Z 325.452,A -85,B 0,C 180,E1 -7515.269,E2 -7515.269} C_VEL
LIN {X 0,Y 467.934,Z 318.482,A -85,B 0,C 180,E1 -7516.131,E2 -7516.131} C_VEL
LIN {X 0,Y 468.191,Z 310.691,A -85,B 0,C 180,E1 -7516.92,E2 -7516.92} C_VEL
LIN {X 0,Y 468.558,Z 300.787,A -85,B 0,C 180,E1 -7517.723,E2 -7517.723} C_VEL
LIN {X 0,Y 468.863,Z 290.463,A -85,B 0,C 180,E1 -7518.347,E2 -7518.347} C_VEL
LIN {X 0,Y 468.828,Z 281.718,A -85,B 0,C 180,E1 -7518.752,E2 -7518.752} C_VEL
LIN {X 0,Y 466.98,Z 271.563,A -85,B 0,C 180,E1 -7519.144,E2 -7519.144} C_VEL
LIN {X 0,Y 467.033,Z 264.551,A -85,B 0,C 180,E1 -7522.439,E2 -7522.439} C_VEL
LIN {X 0,Y 467.098,Z 257.272,A -85,B 0,C 180,E1 -7525.847,E2 -7525.847} C_VEL
LIN {X 0,Y 467.189,Z 252.241,A -85,B 0,C 180,E1 -7528.23,E2 -7528.23} C_VEL
LIN {X 0,Y 467.252,Z 244.447,A -85,B 0,C 180,E1 -7531.719,E2 -7531.719} C_VEL
LIN {X 0,Y 467.256,Z 236.804,A -85,B 0,C 180,E1 -7535.093,E2 -7535.093} C_VEL
LIN {X 0,Y 467.374,Z 230.276,A -85,B 0,C 180,E1 -7537.918,E2 -7537.918} C_VEL
LIN {X 0,Y 467.614,Z 230.239,A -85,B 0,C 180,E1 -7540.692,E2 -7540.692} C_VEL
LIN {X 0,Y 467.652,Z 230.234,A -85,B 0,C 180,E1 -7544.115,E2 -7544.115} C_VEL
LIN {X 0,Y 467.657,Z 230.234,A -85,B 0,C 180,E1 -7547.642,E2 -7547.642} C_VEL
LIN {X 0,Y 467.667,Z 230.234,A -85,B 0,C 180,E1 -7550.485,E2 -7550.485} C_VEL
LIN {X 0,Y 467.66,Z 230.235,A -85,B 0,C 180,E1 -7553.095,E2 -7553.095} C_VEL
LIN {X 0,Y 467.719,Z 230.225,A -85,B 0,C 180,E1 -7554.827,E2 -7554.827} C_VEL
LIN {X 0,Y 467.862,Z 230.208,A -85,B 0,C 180,E1 -7557.417,E2 -7557.417} C_VEL
LIN {X 0,Y 467.886,Z 230.205,A -85,B 0,C 180,E1 -7560,E2 -7560} C_VEL
LIN {X 0,Y 467.862,Z 230.21,A -85,B 0,C 180,E1 -7562.583,E2 -7562.583} C_VEL
LIN {X 0,Y 467.724,Z 230.225,A -85,B 0,C 180,E1 -7566.038,E2 -7566.038} C_VEL
LIN {X 0,Y 467.683,Z 230.23,A -85,B 0,C 180,E1 -7568.643,E2 -7568.643} C_VEL
LIN {X 0,Y 467.659,Z 230.234,A -85,B 0,C 180,E1 -7572.145,E2 -7572.145} C_VEL
LIN {X 0,Y 467.642,Z 230.234,A -85,B 0,C 180,E1 -7575.695,E2 -7575.695} C_VEL
LIN {X 0,Y 467.616,Z 230.237,A -85,B 0,C 180,E1 -7578.763,E2 -7578.763} C_VEL
LIN {X 0,Y 467.583,Z 230.242,A -85,B 0,C 180,E1 -7581.268,E2 -7581.268} C_VEL
LIN {X 0,Y 467.559,Z 230.245,A -85,B 0,C 180,E1 -7583.944,E2 -7583.944} C_VEL
LIN {X 0,Y 467.589,Z 230.239,A -85,B 0,C 180,E1 -7586.802,E2 -7586.802} C_VEL
LIN {X 0,Y 467.555,Z 230.245,A -85,B 0,C 180,E1 -7589.738,E2 -7589.738} C_VEL
LIN {X 0,Y 467.581,Z 230.241,A -85,B 0,C 180,E1 -7592.759,E2 -7592.759} C_VEL
LIN {X 0,Y 467.555,Z 230.247,A -85,B 0,C 180,E1 -7595.89,E2 -7595.89} C_VEL
LIN {X 0,Y 467.584,Z 230.243,A -85,B 0,C 180,E1 -7599.145,E2 -7599.145} C_VEL
LIN {X 0,Y 467.588,Z 230.241,A -85,B 0,C 180,E1 -7602.567,E2 -7602.567} C_VEL
LIN {X 0,Y 467.568,Z 230.245,A -85,B 0,C 180,E1 -7605.053,E2 -7605.053} C_VEL
LIN {X 0,Y 467.591,Z 230.243,A -85,B 0,C 180,E1 -7607.44,E2 -7607.44} C_VEL
LIN {X 0,Y 467.6,Z 230.275,A -85,B 0,C 180,E1 -7609.596,E2 -7609.596} C_VEL
LIN {X 0,Y 468.785,Z 237.069,A -85,B 0,C 180,E1 -7612.615,E2 -7612.615} C_VEL
LIN {X 0,Y 469.212,Z 240.939,A -85,B 0,C 180,E1 -7614.257,E2 -7614.257} C_VEL
LIN {X 0,Y 469.012,Z 246.079,A -85,B 0,C 180,E1 -7616.328,E2 -7616.328} C_VEL
LIN {X 0,Y 468.534,Z 253.788,A -85,B 0,C 180,E1 -7619.336,E2 -7619.336} C_VEL
LIN {X 0,Y 468.102,Z 261.754,A -85,B 0,C 180,E1 -7622.352,E2 -7622.352} C_VEL
LIN {X 0,Y 467.761,Z 270.55,A -85,B 0,C 180,E1 -7625.595,E2 -7625.595} C_VEL
LIN {X 0,Y 467.41,Z 279.599,A -85,B 0,C 180,E1 -7628.847,E2 -7628.847} C_VEL
LIN {X 0,Y 467.151,Z 288.673,A -85,B 0,C 180,E1 -7632.037,E2 -7632.037} C_VEL
LIN {X 0,Y 467.014,Z 296.194,A -85,B 0,C 180,E1 -7634.645,E2 -7634.645} C_VEL
LIN {X 0,Y 469.077,Z 311.512,A -85,B 0,C 180,E1 -7635.168,E2 -7635.168} C_VEL
LIN {X 0,Y 469.683,Z 318.817,A -85,B 0,C 180,E1 -7635.485,E2 -7635.485} C_VEL
LIN {X 0,Y 469.201,Z 331.465,A -85,B 0,C 180,E1 -7636.134,E2 -7636.134} C_VEL
LIN {X 0,Y 468.704,Z 342.735,A -85,B 0,C 180,E1 -7636.892,E2 -7636.892} C_VEL
LIN {X 0,Y 468.203,Z 354.273,A -85,B 0,C 180,E1 -7637.869,E2 -7637.869} C_VEL
LIN {X 0,Y 467.756,Z 364.566,A -85,B 0,C 180,E1 -7638.956,E2 -7638.956} C_VEL
LIN {X 0,Y 467.342,Z 374.454,A -85,B 0,C 180,E1 -7640.26,E2 -7640.26} C_VEL
LIN {X 0,Y 467.039,Z 382.411,A -85,B 0,C 180,E1 -7641.563,E2 -7641.563} C_VEL
LIN {X 0,Y 466.933,Z 387.807,A -85,B 0,C 180,E1 -7642.65,E2 -7642.65} C_VEL
LIN {X 0,Y 466.752,Z 393.069,A -85,B 0,C 180,E1 -7643.95,E2 -7643.95} C_VEL
LIN {X 0,Y 466.692,Z 397.142,A -85,B 0,C 180,E1 -7645.249,E2 -7645.249} C_VEL
LIN {X 0,Y 466.729,Z 400.142,A -85,B 0,C 180,E1 -7646.547,E2 -7646.547} C_VEL
LIN {X 0,Y 466.701,Z 401.576,A -85,B 0,C 180,E1 -7647.411,E2 -7647.411} C_VEL
LIN {X 0,Y 466.693,Z 402.58,A -85,B 0,C 180,E1 -7648.274,E2 -7648.274} C_VEL
LIN {X 0,Y 466.623,Z 403.181,A -85,B 0,C 180,E1 -7649.137,E2 -7649.137} C_VEL
LIN {X 0,Y 466.607,Z 403.382,A -85,B 0,C 180,E1 -7650,E2 -7650} C_VEL
LIN {X 0,Y 466.623,Z 403.136,A -85,B 0,C 180,E1 -7650.863,E2 -7650.863} C_VEL
LIN {X 0,Y 466.693,Z 402.483,A -85,B 0,C 180,E1 -7651.726,E2 -7651.726} C_VEL
LIN {X 0,Y 466.701,Z 401.422,A -85,B 0,C 180,E1 -7652.589,E2 -7652.589} C_VEL
LIN {X 0,Y 466.731,Z 399.945,A -85,B 0,C 180,E1 -7653.453,E2 -7653.453} C_VEL
LIN {X 0,Y 466.697,Z 396.856,A -85,B 0,C 180,E1 -7654.751,E2 -7654.751} C_VEL
LIN {X 0,Y 466.742,Z 392.691,A -85,B 0,C 180,E1 -7656.051,E2 -7656.051} C_VEL
LIN {X 0,Y 466.924,Z 386.305,A -85,B 0,C 180,E1 -7657.568,E2 -7657.568} C_VEL
LIN {X 0,Y 467.098,Z 379.36,A -85,B 0,C 180,E1 -7658.872,E2 -7658.872} C_VEL
LIN {X 0,Y 467.407,Z 370.762,A -85,B 0,C 180,E1 -7660.176,E2 -7660.176} C_VEL
LIN {X 0,Y 467.827,Z 361.943,A -85,B 0,C 180,E1 -7661.262,E2 -7661.262} C_VEL
LIN {X 0,Y 468.259,Z 350.703,A -85,B 0,C 180,E1 -7662.395,E2 -7662.395} C_VEL
LIN {X 0,Y 468.786,Z 339.108,A -85,B 0,C 180,E1 -7663.327,E2 -7663.327} C_VEL
LIN {X 0,Y 469.367,Z 327.142,A -85,B 0,C 180,E1 -7664.083,E2 -7664.083} C_VEL
LIN {X 0,Y 469.646,Z 316.232,A -85,B 0,C 180,E1 -7664.627,E2 -7664.627} C_VEL
LIN {X 0,Y 468.245,Z 303.279,A -85,B 0,C 180,E1 -7665.17,E2 -7665.17} C_VEL
LIN {X 0,Y 466.94,Z 294.263,A -85,B 0,C 180,E1 -7665.485,E2 -7665.485} C_VEL
LIN {X 0,Y 467.134,Z 284.22,A -85,B 0,C 180,E1 -7668.902,E2 -7668.902} C_VEL
LIN {X 0,Y 467.391,Z 275.19,A -85,B 0,C 180,E1 -7672.081,E2 -7672.081} C_VEL
LIN {X 0,Y 467.719,Z 265.606,A -85,B 0,C 180,E1 -7675.635,E2 -7675.635} C_VEL
LIN {X 0,Y 468.104,Z 257.859,A -85,B 0,C 180,E1 -7678.714,E2 -7678.714} C_VEL
LIN {X 0,Y 468.649,Z 251.048,A -85,B 0,C 180,E1 -7681.66,E2 -7681.66} C_VEL
LIN {X 0,Y 469.294,Z 245.117,A -85,B 0,C 180,E1 -7684.547,E2 -7684.547} C_VEL
LIN {X 0,Y 469.417,Z 242.402,A -85,B 0,C 180,E1 -7686.053,E2 -7686.053} C_VEL
LIN {X 0,Y 469.174,Z 239.538,A -85,B 0,C 180,E1 -7687.891,E2 -7687.891} C_VEL
LIN {X 0,Y 468.731,Z 236.659,A -85,B 0,C 180,E1 -7690.146,E2 -7690.146} C_VEL
LIN {X 0,Y 468.264,Z 234.275,A -85,B 0,C 180,E1 -7692.657,E2 -7692.657} C_VEL
LIN {X 0,Y 468.02,Z 232.745,A -85,B 0,C 180,E1 -7695.108,E2 -7695.108} C_VEL
LIN {X 0,Y 467.883,Z 231.988,A -85,B 0,C 180,E1 -7697.473,E2 -7697.473} C_VEL
LIN {X 0,Y 467.85,Z 231.883,A -85,B 0,C 180,E1 -7700.007,E2 -7700.007} C_VEL
LIN {X 0,Y 467.954,Z 232.542,A -85,B 0,C 180,E1 -7703.077,E2 -7703.077} C_VEL
LIN {X 0,Y 467.965,Z 233.646,A -85,B 0,C 180,E1 -7705.691,E2 -7705.691} C_VEL
LIN {X 0,Y 467.709,Z 235.541,A -85,B 0,C 180,E1 -7708.927,E2 -7708.927} C_VEL
LIN {X 0,Y 467.528,Z 237.159,A -85,B 0,C 180,E1 -7711.247,E2 -7711.247} C_VEL
LIN {X 0,Y 467.391,Z 239.605,A -85,B 0,C 180,E1 -7714.45,E2 -7714.45} C_VEL
LIN {X 0,Y 467.267,Z 241.702,A -85,B 0,C 180,E1 -7716.98,E2 -7716.98} C_VEL
LIN {X 0,Y 467.12,Z 244.137,A -85,B 0,C 180,E1 -7719.754,E2 -7719.754} C_VEL
LIN {X 0,Y 467.08,Z 246.642,A -85,B 0,C 180,E1 -7722.486,E2 -7722.486} C_VEL
LIN {X 0,Y 467.028,Z 249.215,A -85,B 0,C 180,E1 -7725.178,E2 -7725.178} C_VEL
LIN {X 0,Y 467.015,Z 249.707,A -85,B 0,C 180,E1 -7725.678,E2 -7725.678} C_VEL
LIN {X 0,Y 470.277,Z 262.856,A -85,B 0,C 180,E1 -7726.262,E2 -7726.262} C_VEL
LIN {X 0,Y 470.082,Z 273.999,A -85,B 0,C 180,E1 -7726.783,E2 -7726.783} C_VEL
LIN {X 0,Y 469.698,Z 285.456,A -85,B 0,C 180,E1 -7727.469,E2 -7727.469} C_VEL
LIN {X 0,Y 469.127,Z 296.755,A -85,B 0,C 180,E1 -7728.332,E2 -7728.332} C_VEL
LIN {X 0,Y 468.604,Z 308.058,A -85,B 0,C 180,E1 -7729.413,E2 -7729.413} C_VEL
LIN {X 0,Y 468.224,Z 317.148,A -85,B 0,C 180,E1 -7730.496,E2 -7730.496} C_VEL
LIN {X 0,Y 467.716,Z 325.989,A -85,B 0,C 180,E1 -7731.793,E2 -7731.793} C_VEL
LIN {X 0,Y 467.412,Z 333.706,A -85,B 0,C 180,E1 -7733.214,E2 -7733.214} C_VEL
LIN {X 0,Y 467.189,Z 338.806,A -85,B 0,C 180,E1 -7734.389,E2 -7734.389} C_VEL
LIN {X 0,Y 467.017,Z 343.271,A -85,B 0,C 180,E1 -7735.685,E2 -7735.685} C_VEL
LIN {X 0,Y 467.04,Z 345.606,A -85,B 0,C 180,E1 -7736.549,E2 -7736.549} C_VEL
LIN {X 0,Y 466.86,Z 347.526,A -85,B 0,C 180,E1 -7737.412,E2 -7737.412} C_VEL
LIN {X 0,Y 466.71,Z 349.027,A -85,B 0,C 180,E1 -7738.274,E2 -7738.274} C_VEL
LIN {X 0,Y 466.636,Z 350.07,A -85,B 0,C 180,E1 -7739.137,E2 -7739.137} C_VEL
LIN {X 0,Y 466.63,Z 350.956,A -85,B 0,C 180,E1 -7740.863,E2 -7740.863} C_VEL
LIN {X 0,Y 466.7,Z 350.809,A -85,B 0,C 180,E1 -7741.726,E2 -7741.726} C_VEL
LIN {X 0,Y 466.776,Z 350.221,A -85,B 0,C 180,E1 -7742.589,E2 -7742.589} C_VEL
LIN {X 0,Y 466.811,Z 349.237,A -85,B 0,C 180,E1 -7743.453,E2 -7743.453} C_VEL
LIN {X 0,Y 466.805,Z 347.86,A -85,B 0,C 180,E1 -7744.317,E2 -7744.317} C_VEL
LIN {X 0,Y 466.899,Z 344.956,A -85,B 0,C 180,E1 -7745.615,E2 -7745.615} C_VEL
LIN {X 0,Y 466.956,Z 341.012,A -85,B 0,C 180,E1 -7746.916,E2 -7746.916} C_VEL
LIN {X 0,Y 467.238,Z 334.934,A -85,B 0,C 180,E1 -7748.433,E2 -7748.433} C_VEL
LIN {X 0,Y 467.501,Z 328.255,A -85,B 0,C 180,E1 -7749.737,E2 -7749.737} C_VEL
LIN {X 0,Y 467.866,Z 319.964,A -85,B 0,C 180,E1 -7751.042,E2 -7751.042} C_VEL
LIN {X 0,Y 468.341,Z 310.32,A -85,B 0,C 180,E1 -7752.259,E2 -7752.259} C_VEL
LIN {X 0,Y 468.684,Z 301.023,A -85,B 0,C 180,E1 -7753.219,E2 -7753.219} C_VEL
LIN {X 0,Y 469.239,Z 289.307,A -85,B 0,C 180,E1 -7754.197,E2 -7754.197} C_VEL
LIN {X 0,Y 469.717,Z 277.657,A -85,B 0,C 180,E1 -7754.957,E2 -7754.957} C_VEL
LIN {X 0,Y 470.04,Z 264.533,A -85,B 0,C 180,E1 -7755.613,E2 -7755.613} C_VEL
LIN {X 0,Y 469.614,Z 260.343,A -85,B 0,C 180,E1 -7755.795,E2 -7755.795} C_VEL
LIN {X 0,Y 466.761,Z 247.461,A -85,B 0,C 180,E1 -7756.32,E2 -7756.32} C_VEL
LIN {X 0,Y 466.792,Z 244.034,A -85,B 0,C 180,E1 -7759.344,E2 -7759.344} C_VEL
LIN {X 0,Y 466.803,Z 240.935,A -85,B 0,C 180,E1 -7762.11,E2 -7762.11} C_VEL
LIN {X 0,Y 466.918,Z 236.794,A -85,B 0,C 180,E1 -7765.881,E2 -7765.881} C_VEL
LIN {X 0,Y 466.949,Z 233.644,A -85,B 0,C 180,E1 -7768.792,E2 -7768.792} C_VEL
LIN {X 0,Y 466.978,Z 230.453,A -85,B 0,C 180,E1 -7771.786,E2 -7771.786} C_VEL
LIN {X 0,Y 467.363,Z 230.272,A -85,B 0,C 180,E1 -7774.85,E2 -7774.85} C_VEL
LIN {X 0,Y 467.509,Z 230.249,A -85,B 0,C 180,E1 -7777.179,E2 -7777.179} C_VEL
LIN {X 0,Y 467.575,Z 230.242,A -85,B 0,C 180,E1 -7780.265,E2 -7780.265} C_VEL
LIN {X 0,Y 467.553,Z 230.245,A -85,B 0,C 180,E1 -7783.745,E2 -7783.745} C_VEL
LIN {X 0,Y 467.55,Z 230.243,A -85,B 0,C 180,E1 -7786.254,E2 -7786.254} C_VEL
LIN {X 0,Y 467.56,Z 230.242,A -85,B 0,C 180,E1 -7789.733,E2 -7789.733} C_VEL
LIN {X 0,Y 467.517,Z 230.253,A -85,B 0,C 180,E1 -7792.819,E2 -7792.819} C_VEL
LIN {X 0,Y 467.578,Z 230.238,A -85,B 0,C 180,E1 -7795.76,E2 -7795.76} C_VEL
LIN {X 0,Y 467.571,Z 230.241,A -85,B 0,C 180,E1 -7798.955,E2 -7798.955} C_VEL
LIN {X 0,Y 467.608,Z 230.239,A -85,B 0,C 180,E1 -7802.469,E2 -7802.469} C_VEL
LIN {X 0,Y 467.588,Z 230.24,A -85,B 0,C 180,E1 -7805.111,E2 -7805.111} C_VEL
LIN {X 0,Y 467.539,Z 230.248,A -85,B 0,C 180,E1 -7807.926,E2 -7807.926} C_VEL
LIN {X 0,Y 467.615,Z 230.237,A -85,B 0,C 180,E1 -7810.023,E2 -7810.023} C_VEL
LIN {X 0,Y 466.931,Z 230.323,A -85,B 0,C 180,E1 -7810.742,E2 -7810.742} C_VEL
LIN {X 0,Y 464.052,Z 230.681,A -85,B 0,C 180,E1 -7811.909,E2 -7811.909} C_VEL
LIN {X 0,Y 461.647,Z 230.982,A -85,B 0,C 180,E1 -7812.85,E2 -7812.85} C_VEL
LIN {X 0,Y 460.65,Z 231.106,A -85,B 0,C 180,E1 -7813.577,E2 -7813.577} C_VEL
LIN {X 0,Y 460.587,Z 231.111,A -85,B 0,C 180,E1 -7813.823,E2 -7813.823} C_VEL
LIN {X 0,Y 460.545,Z 231.119,A -85,B 0,C 180,E1 -7816.767,E2 -7816.767} C_VEL
LIN {X 0,Y 460.576,Z 231.112,A -85,B 0,C 180,E1 -7819.449,E2 -7819.449} C_VEL
LIN {X 0,Y 460.662,Z 231.103,A -85,B 0,C 180,E1 -7822.598,E2 -7822.598} C_VEL
LIN {X 0,Y 460.671,Z 231.1,A -85,B 0,C 180,E1 -7824.748,E2 -7824.748} C_VEL
LIN {X 0,Y 460.757,Z 231.09,A -85,B 0,C 180,E1 -7827.377,E2 -7827.377} C_VEL
LIN {X 0,Y 460.826,Z 231.083,A -85,B 0,C 180,E1 -7830,E2 -7830} C_VEL
LIN {X 0,Y 460.794,Z 231.084,A -85,B 0,C 180,E1 -7832.622,E2 -7832.622} C_VEL
LIN {X 0,Y 460.348,Z 231.225,A -85,B 0,C 180,E1 -7835.86,E2 -7835.86} C_VEL
LIN {X 0,Y 460.201,Z 237.552,A -85,B 0,C 180,E1 -7838.784,E2 -7838.784} C_VEL
LIN {X 0,Y 460.201,Z 245.188,A -85,B 0,C 180,E1 -7842.345,E2 -7842.345} C_VEL
LIN {X 0,Y 460.095,Z 252.46,A -85,B 0,C 180,E1 -7845.775,E2 -7845.775} C_VEL
LIN {X 0,Y 460.009,Z 258.687,A -85,B 0,C 180,E1 -7848.714,E2 -7848.714} C_VEL
LIN {X 0,Y 459.861,Z 265.575,A -85,B 0,C 180,E1 -7851.989,E2 -7851.989} C_VEL
LIN {X 0,Y 459.906,Z 271.483,A -85,B 0,C 180,E1 -7854.789,E2 -7854.789} C_VEL
LIN {X 0,Y 461.963,Z 283.822,A -85,B 0,C 180,E1 -7855.273,E2 -7855.273} C_VEL
LIN {X 0,Y 461.723,Z 294.588,A -85,B 0,C 180,E1 -7855.83,E2 -7855.83} C_VEL
LIN {X 0,Y 461.418,Z 303.768,A -85,B 0,C 180,E1 -7856.456,E2 -7856.456} C_VEL
LIN {X 0,Y 461.098,Z 312.533,A -85,B 0,C 180,E1 -7857.21,E2 -7857.21} C_VEL
LIN {X 0,Y 460.743,Z 321.842,A -85,B 0,C 180,E1 -7858.22,E2 -7858.22} C_VEL
LIN {X 0,Y 460.452,Z 329.132,A -85,B 0,C 180,E1 -7859.237,E2 -7859.237} C_VEL
LIN {X 0,Y 460.195,Z 335.099,A -85,B 0,C 180,E1 -7860.263,E2 -7860.263} C_VEL
LIN {X 0,Y 459.998,Z 339.953,A -85,B 0,C 180,E1 -7861.296,E2 -7861.296} C_VEL
LIN {X 0,Y 459.815,Z 343.859,A -85,B 0,C 180,E1 -7862.341,E2 -7862.341} C_VEL
LIN {X 0,Y 459.737,Z 346.878,A -85,B 0,C 180,E1 -7863.39,E2 -7863.39} C_VEL
LIN {X 0,Y 459.643,Z 349.112,A -85,B 0,C 180,E1 -7864.453,E2 -7864.453} C_VEL
LIN {X 0,Y 459.555,Z 350.931,A -85,B 0,C 180,E1 -7865.851,E2 -7865.851} C_VEL
LIN {X 0,Y 459.499,Z 351.367,A -85,B 0,C 180,E1 -7867.313,E2 -7867.313} C_VEL
LIN {X 0,Y 459.574,Z 350.37,A -85,B 0,C 180,E1 -7868.828,E2 -7868.828} C_VEL
LIN {X 0,Y 459.692,Z 348.331,A -85,B 0,C 180,E1 -7870.144,E2 -7870.144} C_VEL
LIN {X 0,Y 459.845,Z 344.895,A -85,B 0,C 180,E1 -7871.506,E2 -7871.506} C_VEL
LIN {X 0,Y 460.014,Z 341.295,A -85,B 0,C 180,E1 -7872.541,E2 -7872.541} C_VEL
LIN {X 0,Y 460.195,Z 335.687,A -85,B 0,C 180,E1 -7873.779,E2 -7873.779} C_VEL
LIN {X 0,Y 460.422,Z 331.109,A -85,B 0,C 180,E1 -7874.6,E2 -7874.6} C_VEL
LIN {X 0,Y 460.708,Z 324.521,A -85,B 0,C 180,E1 -7875.576,E2 -7875.576} C_VEL
LIN {X 0,Y 460.986,Z 317.749,A -85,B 0,C 180,E1 -7876.4,E2 -7876.4} C_VEL
LIN {X 0,Y 461.387,Z 308.608,A -85,B 0,C 180,E1 -7877.304,E2 -7877.304} C_VEL
LIN {X 0,Y 461.65,Z 299.109,A -85,B 0,C 180,E1 -7878.03,E2 -7878.03} C_VEL
LIN {X 0,Y 461.964,Z 289.109,A -85,B 0,C 180,E1 -7878.61,E2 -7878.61} C_VEL
LIN {X 0,Y 462.071,Z 284.249,A -85,B 0,C 180,E1 -7878.847,E2 -7878.847} C_VEL
LIN {X 0,Y 460.177,Z 273.316,A -85,B 0,C 180,E1 -7879.285,E2 -7879.285} C_VEL
LIN {X 0,Y 459.926,Z 271.877,A -85,B 0,C 180,E1 -7879.359,E2 -7879.359} C_VEL
LIN {X 0,Y 459.982,Z 265.583,A -85,B 0,C 180,E1 -7882.327,E2 -7882.327} C_VEL
LIN {X 0,Y 460.054,Z 258.664,A -85,B 0,C 180,E1 -7885.582,E2 -7885.582} C_VEL
LIN {X 0,Y 460.125,Z 253.034,A -85,B 0,C 180,E1 -7888.2,E2 -7888.2} C_VEL
LIN {X 0,Y 460.189,Z 246.417,A -85,B 0,C 180,E1 -7891.245,E2 -7891.245} C_VEL
LIN {X 0,Y 460.232,Z 238.636,A -85,B 0,C 180,E1 -7894.686,E2 -7894.686} C_VEL
LIN {X 0,Y 460.354,Z 231.15,A -85,B 0,C 180,E1 -7898.035,E2 -7898.035} C_VEL
LIN {X 0,Y 460.553,Z 231.119,A -85,B 0,C 180,E1 -7900.384,E2 -7900.384} C_VEL
LIN {X 0,Y 460.562,Z 231.118,A -85,B 0,C 180,E1 -7903.146,E2 -7903.146} C_VEL
LIN {X 0,Y 460.557,Z 231.12,A -85,B 0,C 180,E1 -7905.868,E2 -7905.868} C_VEL
LIN {X 0,Y 460.614,Z 231.112,A -85,B 0,C 180,E1 -7908.559,E2 -7908.559} C_VEL
LIN {X 0,Y 460.67,Z 231.104,A -85,B 0,C 180,E1 -7912.108,E2 -7912.108} C_VEL
LIN {X 0,Y 460.69,Z 231.101,A -85,B 0,C 180,E1 -7914.748,E2 -7914.748} C_VEL
LIN {X 0,Y 460.803,Z 231.087,A -85,B 0,C 180,E1 -7917.377,E2 -7917.377} C_VEL
LIN {X 0,Y 460.856,Z 231.081,A -85,B 0,C 180,E1 -7920,E2 -7920} C_VEL
LIN {X 0,Y 460.803,Z 231.089,A -85,B 0,C 180,E1 -7922.622,E2 -7922.622} C_VEL
LIN {X 0,Y 460.688,Z 231.102,A -85,B 0,C 180,E1 -7926.13,E2 -7926.13} C_VEL
LIN {X 0,Y 460.63,Z 231.108,A -85,B 0,C 180,E1 -7928.776,E2 -7928.776} C_VEL
LIN {X 0,Y 460.616,Z 231.11,A -85,B 0,C 180,E1 -7932.445,E2 -7932.445} C_VEL
LIN {X 0,Y 460.603,Z 231.109,A -85,B 0,C 180,E1 -7935.997,E2 -7935.997} C_VEL
LIN {X 0,Y 460.571,Z 231.115,A -85,B 0,C 180,E1 -7939.615,E2 -7939.615} C_VEL
LIN {X 0,Y 460.513,Z 231.123,A -85,B 0,C 180,E1 -7942.429,E2 -7942.429} C_VEL
LIN {X 0,Y 460.548,Z 231.118,A -85,B 0,C 180,E1 -7945.796,E2 -7945.796} C_VEL
LIN {X 0,Y 460.552,Z 231.118,A -85,B 0,C 180,E1 -7948.233,E2 -7948.233} C_VEL
LIN {X 0,Y 460.522,Z 231.121,A -85,B 0,C 180,E1 -7951.283,E2 -7951.283} C_VEL
LIN {X 0,Y 460.525,Z 231.121,A -85,B 0,C 180,E1 -7954.504,E2 -7954.504} C_VEL
LIN {X 0,Y 460.503,Z 231.122,A -85,B 0,C 180,E1 -7957.623,E2 -7957.623} C_VEL
LIN {X 0,Y 460.544,Z 231.118,A -85,B 0,C 180,E1 -7960.269,E2 -7960.269} C_VEL
LIN {X 0,Y 460.5,Z 231.124,A -85,B 0,C 180,E1 -7963.375,E2 -7963.375} C_VEL
LIN {X 0,Y 460.5,Z 231.127,A -85,B 0,C 180,E1 -7966.625,E2 -7966.625} C_VEL
LIN {X 0,Y 460.571,Z 231.239,A -85,B 0,C 180,E1 -7969.391,E2 -7969.391} C_VEL
LIN {X 0,Y 461.781,Z 238.104,A -85,B 0,C 180,E1 -7972.499,E2 -7972.499} C_VEL
LIN {X 0,Y 462.217,Z 242.086,A -85,B 0,C 180,E1 -7974.209,E2 -7974.209} C_VEL
LIN {X 0,Y 462.004,Z 247.123,A -85,B 0,C 180,E1 -7976.273,E2 -7976.273} C_VEL
LIN {X 0,Y 461.524,Z 254.816,A -85,B 0,C 180,E1 -7979.327,E2 -7979.327} C_VEL
LIN {X 0,Y 461.104,Z 262.096,A -85,B 0,C 180,E1 -7982.131,E2 -7982.131} C_VEL
LIN {X 0,Y 460.747,Z 270.268,A -85,B 0,C 180,E1 -7985.199,E2 -7985.199} C_VEL
LIN {X 0,Y 460.369,Z 279.297,A -85,B 0,C 180,E1 -7988.507,E2 -7988.507} C_VEL
LIN {X 0,Y 460.156,Z 287.043,A -85,B 0,C 180,E1 -7991.293,E2 -7991.293} C_VEL
LIN {X 0,Y 459.947,Z 295.897,A -85,B 0,C 180,E1 -7994.432,E2 -7994.432} C_VEL
LIN {X 0,Y 462.02,Z 310.925,A -85,B 0,C 180,E1 -7994.95,E2 -7994.95} C_VEL
LIN {X 0,Y 462.744,Z 319.22,A -85,B 0,C 180,E1 -7995.319,E2 -7995.319} C_VEL
LIN {X 0,Y 462.267,Z 330.724,A -85,B 0,C 180,E1 -7995.921,E2 -7995.921} C_VEL
LIN {X 0,Y 461.756,Z 342.076,A -85,B 0,C 180,E1 -7996.691,E2 -7996.691} C_VEL
LIN {X 0,Y 461.203,Z 353.653,A -85,B 0,C 180,E1 -7997.682,E2 -7997.682} C_VEL
LIN {X 0,Y 460.744,Z 364.002,A -85,B 0,C 180,E1 -7998.786,E2 -7998.786} C_VEL
LIN {X 0,Y 460.293,Z 373.918,A -85,B 0,C 180,E1 -8000.109,E2 -8000.109} C_VEL
LIN {X 0,Y 459.985,Z 381.911,A -85,B 0,C 180,E1 -8001.433,E2 -8001.433} C_VEL
LIN {X 0,Y 459.84,Z 387.323,A -85,B 0,C 180,E1 -8002.536,E2 -8002.536} C_VEL
LIN {X 0,Y 459.661,Z 392.609,A -85,B 0,C 180,E1 -8003.856,E2 -8003.856} C_VEL
LIN {X 0,Y 459.623,Z 396.703,A -85,B 0,C 180,E1 -8005.176,E2 -8005.176} C_VEL
LIN {X 0,Y 459.626,Z 399.715,A -85,B 0,C 180,E1 -8006.494,E2 -8006.494} C_VEL
LIN {X 0,Y 459.621,Z 401.163,A -85,B 0,C 180,E1 -8007.371,E2 -8007.371} C_VEL
LIN {X 0,Y 459.63,Z 402.173,A -85,B 0,C 180,E1 -8008.248,E2 -8008.248} C_VEL
LIN {X 0,Y 459.556,Z 402.776,A -85,B 0,C 180,E1 -8009.124,E2 -8009.124} C_VEL
LIN {X 0,Y 459.538,Z 402.98,A -85,B 0,C 180,E1 -8010,E2 -8010} C_VEL
LIN {X 0,Y 459.557,Z 402.739,A -85,B 0,C 180,E1 -8010.876,E2 -8010.876} C_VEL
LIN {X 0,Y 459.614,Z 402.083,A -85,B 0,C 180,E1 -8011.753,E2 -8011.753} C_VEL
LIN {X 0,Y 459.622,Z 401.022,A -85,B 0,C 180,E1 -8012.629,E2 -8012.629} C_VEL
LIN {X 0,Y 459.628,Z 399.543,A -85,B 0,C 180,E1 -8013.507,E2 -8013.507} C_VEL
LIN {X 0,Y 459.627,Z 396.453,A -85,B 0,C 180,E1 -8014.824,E2 -8014.824} C_VEL
LIN {X 0,Y 459.714,Z 391.207,A -85,B 0,C 180,E1 -8016.431,E2 -8016.431} C_VEL
LIN {X 0,Y 459.884,Z 384.85,A -85,B 0,C 180,E1 -8017.906,E2 -8017.906} C_VEL
LIN {X 0,Y 460.101,Z 377.674,A -85,B 0,C 180,E1 -8019.23,E2 -8019.23} C_VEL
LIN {X 0,Y 460.446,Z 368.719,A -85,B 0,C 180,E1 -8020.554,E2 -8020.554} C_VEL
LIN {X 0,Y 460.954,Z 358.615,A -85,B 0,C 180,E1 -8021.767,E2 -8021.767} C_VEL
LIN {X 0,Y 461.335,Z 348.462,A -85,B 0,C 180,E1 -8022.759,E2 -8022.759} C_VEL
LIN {X 0,Y 462.001,Z 335.766,A -85,B 0,C 180,E1 -8023.75,E2 -8023.75} C_VEL
LIN {X 0,Y 462.645,Z 323.057,A -85,B 0,C 180,E1 -8024.516,E2 -8024.516} C_VEL
LIN {X 0,Y 462.619,Z 316.303,A -85,B 0,C 180,E1 -8024.854,E2 -8024.854} C_VEL
LIN {X 0,Y 461.259,Z 302.942,A -85,B 0,C 180,E1 -8025.434,E2 -8025.434} C_VEL
LIN {X 0,Y 459.854,Z 293.782,A -85,B 0,C 180,E1 -8025.76,E2 -8025.76} C_VEL
LIN {X 0,Y 460.081,Z 283.981,A -85,B 0,C 180,E1 -8029.173,E2 -8029.173} C_VEL
LIN {X 0,Y 460.352,Z 274.948,A -85,B 0,C 180,E1 -8032.437,E2 -8032.437} C_VEL
LIN {X 0,Y 460.695,Z 266.02,A -85,B 0,C 180,E1 -8035.834,E2 -8035.834} C_VEL
LIN {X 0,Y 461.072,Z 259.01,A -85,B 0,C 180,E1 -8038.695,E2 -8038.695} C_VEL
LIN {X 0,Y 461.616,Z 252.647,A -85,B 0,C 180,E1 -8041.506,E2 -8041.506} C_VEL
LIN {X 0,Y 462.257,Z 247.101,A -85,B 0,C 180,E1 -8044.232,E2 -8044.232} C_VEL
LIN {X 0,Y 462.441,Z 243.367,A -85,B 0,C 180,E1 -8046.35,E2 -8046.35} C_VEL
LIN {X 0,Y 462.101,Z 240.118,A -85,B 0,C 180,E1 -8048.577,E2 -8048.577} C_VEL
LIN {X 0,Y 461.647,Z 237.439,A -85,B 0,C 180,E1 -8050.891,E2 -8050.891} C_VEL
LIN {X 0,Y 461.273,Z 235.386,A -85,B 0,C 180,E1 -8053.285,E2 -8053.285} C_VEL
LIN {X 0,Y 461.04,Z 234.024,A -85,B 0,C 180,E1 -8055.763,E2 -8055.763} C_VEL
LIN {X 0,Y 460.893,Z 233.332,A -85,B 0,C 180,E1 -8059.028,E2 -8059.028} C_VEL
LIN {X 0,Y 460.933,Z 233.481,A -85,B 0,C 180,E1 -8061.307,E2 -8061.307} C_VEL
LIN {X 0,Y 460.98,Z 234.441,A -85,B 0,C 180,E1 -8064.596,E2 -8064.596} C_VEL
LIN {X 0,Y 460.858,Z 235.59,A -85,B 0,C 180,E1 -8067.008,E2 -8067.008} C_VEL
LIN {X 0,Y 460.632,Z 237.244,A -85,B 0,C 180,E1 -8069.769,E2 -8069.769} C_VEL
LIN {X 0,Y 460.447,Z 239.336,A -85,B 0,C 180,E1 -8072.748,E2 -8072.748} C_VEL
LIN {X 0,Y 460.279,Z 241.584,A -85,B 0,C 180,E1 -8075.653,E2 -8075.653} C_VEL
LIN {X 0,Y 460.134,Z 244.128,A -85,B 0,C 180,E1 -8078.703,E2 -8078.703} C_VEL
LIN {X 0,Y 460.094,Z 246.409,A -85,B 0,C 180,E1 -8081.29,E2 -8081.29} C_VEL
LIN {X 0,Y 460.031,Z 249.155,A -85,B 0,C 180,E1 -8084.254,E2 -8084.254} C_VEL
LIN {X 0,Y 459.993,Z 250.256,A -85,B 0,C 180,E1 -8085.398,E2 -8085.398} C_VEL
LIN {X 0,Y 463.481,Z 264.116,A -85,B 0,C 180,E1 -8086.042,E2 -8086.042} C_VEL
LIN {X 0,Y 463.251,Z 275.077,A -85,B 0,C 180,E1 -8086.574,E2 -8086.574} C_VEL
LIN {X 0,Y 462.842,Z 286.472,A -85,B 0,C 180,E1 -8087.281,E2 -8087.281} C_VEL
LIN {X 0,Y 462.242,Z 297.629,A -85,B 0,C 180,E1 -8088.156,E2 -8088.156} C_VEL
LIN {X 0,Y 461.675,Z 308.829,A -85,B 0,C 180,E1 -8089.253,E2 -8089.253} C_VEL
LIN {X 0,Y 461.266,Z 317.827,A -85,B 0,C 180,E1 -8090.352,E2 -8090.352} C_VEL
LIN {X 0,Y 460.733,Z 326.612,A -85,B 0,C 180,E1 -8091.668,E2 -8091.668} C_VEL
LIN {X 0,Y 460.398,Z 333.704,A -85,B 0,C 180,E1 -8092.986,E2 -8092.986} C_VEL
LIN {X 0,Y 460.156,Z 339.353,A -85,B 0,C 180,E1 -8094.303,E2 -8094.303} C_VEL
LIN {X 0,Y 459.974,Z 343.782,A -85,B 0,C 180,E1 -8095.619,E2 -8095.619} C_VEL
LIN {X 0,Y 459.993,Z 346.1,A -85,B 0,C 180,E1 -8096.496,E2 -8096.496} C_VEL
LIN {X 0,Y 459.808,Z 348.004,A -85,B 0,C 180,E1 -8097.372,E2 -8097.372} C_VEL
LIN {X 0,Y 459.649,Z 349.49,A -85,B 0,C 180,E1 -8098.248,E2 -8098.248} C_VEL
LIN {X 0,Y 459.569,Z 350.513,A -85,B 0,C 180,E1 -8099.124,E2 -8099.124} C_VEL
LIN {X 0,Y 459.563,Z 351.368,A -85,B 0,C 180,E1 -8100.876,E2 -8100.876} C_VEL
LIN {X 0,Y 459.638,Z 351.196,A -85,B 0,C 180,E1 -8101.753,E2 -8101.753} C_VEL
LIN {X 0,Y 459.693,Z 350.586,A -85,B 0,C 180,E1 -8102.629,E2 -8102.629} C_VEL
LIN {X 0,Y 459.742,Z 349.584,A -85,B 0,C 180,E1 -8103.506,E2 -8103.506} C_VEL
LIN {X 0,Y 459.716,Z 348.186,A -85,B 0,C 180,E1 -8104.384,E2 -8104.384} C_VEL
LIN {X 0,Y 459.85,Z 345.242,A -85,B 0,C 180,E1 -8105.701,E2 -8105.701} C_VEL
LIN {X 0,Y 459.914,Z 341.255,A -85,B 0,C 180,E1 -8107.022,E2 -8107.022} C_VEL
LIN {X 0,Y 460.191,Z 335.107,A -85,B 0,C 180,E1 -8108.563,E2 -8108.563} C_VEL
LIN {X 0,Y 460.467,Z 328.372,A -85,B 0,C 180,E1 -8109.887,E2 -8109.887} C_VEL
LIN {X 0,Y 460.877,Z 320.017,A -85,B 0,C 180,E1 -8111.211,E2 -8111.211} C_VEL
LIN {X 0,Y 461.34,Z 311.443,A -85,B 0,C 180,E1 -8112.314,E2 -8112.314} C_VEL
LIN {X 0,Y 461.695,Z 302.058,A -85,B 0,C 180,E1 -8113.311,E2 -8113.311} C_VEL
LIN {X 0,Y 462.252,Z 290.486,A -85,B 0,C 180,E1 -8114.304,E2 -8114.304} C_VEL
LIN {X 0,Y 462.766,Z 279.185,A -85,B 0,C 180,E1 -8115.073,E2 -8115.073} C_VEL
LIN {X 0,Y 463.114,Z 265.789,A -85,B 0,C 180,E1 -8115.767,E2 -8115.767} C_VEL
LIN {X 0,Y 462.824,Z 262.005,A -85,B 0,C 180,E1 -8115.938,E2 -8115.938} C_VEL
LIN {X 0,Y 459.735,Z 248.253,A -85,B 0,C 180,E1 -8116.493,E2 -8116.493} C_VEL
LIN {X 0,Y 459.69,Z 247.82,A -85,B 0,C 180,E1 -8116.509,E2 -8116.509} C_VEL
LIN {X 0,Y 459.719,Z 244.268,A -85,B 0,C 180,E1 -8119.653,E2 -8119.653} C_VEL
LIN {X 0,Y 459.717,Z 241.142,A -85,B 0,C 180,E1 -8122.47,E2 -8122.47} C_VEL
LIN {X 0,Y 459.871,Z 237.688,A -85,B 0,C 180,E1 -8125.62,E2 -8125.62} C_VEL
LIN {X 0,Y 459.867,Z 234.836,A -85,B 0,C 180,E1 -8128.279,E2 -8128.279} C_VEL
LIN {X 0,Y 459.902,Z 231.622,A -85,B 0,C 180,E1 -8131.304,E2 -8131.304} C_VEL
LIN {X 0,Y 460.064,Z 231.18,A -85,B 0,C 180,E1 -8132.839,E2 -8132.839} C_VEL
LIN {X 0,Y 460.39,Z 231.141,A -85,B 0,C 180,E1 -8135.457,E2 -8135.457} C_VEL
LIN {X 0,Y 460.515,Z 231.121,A -85,B 0,C 180,E1 -8138.735,E2 -8138.735} C_VEL
LIN {X 0,Y 460.522,Z 231.123,A -85,B 0,C 180,E1 -8141.6,E2 -8141.6} C_VEL
LIN {X 0,Y 460.516,Z 231.12,A -85,B 0,C 180,E1 -8144.589,E2 -8144.589} C_VEL
LIN {X 0,Y 460.494,Z 231.123,A -85,B 0,C 180,E1 -8147.815,E2 -8147.815} C_VEL
LIN {X 0,Y 460.512,Z 231.119,A -85,B 0,C 180,E1 -8150.135,E2 -8150.135} C_VEL
LIN {X 0,Y 460.461,Z 231.125,A -85,B 0,C 180,E1 -8153.469,E2 -8153.469} C_VEL
LIN {X 0,Y 460.52,Z 231.123,A -85,B 0,C 180,E1 -8156.674,E2 -8156.674} C_VEL
LIN {X 0,Y 460.511,Z 231.121,A -85,B 0,C 180,E1 -8159.76,E2 -8159.76} C_VEL
LIN {X 0,Y 460.539,Z 231.117,A -85,B 0,C 180,E1 -8162.754,E2 -8162.754} C_VEL
LIN {X 0,Y 460.534,Z 231.119,A -85,B 0,C 180,E1 -8165.667,E2 -8165.667} C_VEL
LIN {X 0,Y 460.526,Z 231.119,A -85,B 0,C 180,E1 -8168.578,E2 -8168.578} C_VEL
LIN {X 0,Y 460.59,Z 231.112,A -85,B 0,C 180,E1 -8171.311,E2 -8171.311} C_VEL
LIN {X 0,Y 460.587,Z 231.111,A -85,B 0,C 180,E1 -8173.823,E2 -8173.823} C_VEL
LIN {X 0,Y 459.972,Z 231.19,A -85,B 0,C 180,E1 -8174.553,E2 -8174.553} C_VEL
LIN {X 0,Y 457.14,Z 231.543,A -85,B 0,C 180,E1 -8175.737,E2 -8175.737} C_VEL
LIN {X 0,Y 454.706,Z 231.846,A -85,B 0,C 180,E1 -8176.692,E2 -8176.692} C_VEL
LIN {X 0,Y 453.648,Z 231.976,A -85,B 0,C 180,E1 -8177.431,E2 -8177.431} C_VEL
LIN {X 0,Y 453.556,Z 231.987,A -85,B 0,C 180,E1 -8177.681,E2 -8177.681} C_VEL
LIN {X 0,Y 453.58,Z 231.984,A -85,B 0,C 180,E1 -8181.086,E2 -8181.086} C_VEL
LIN {X 0,Y 453.631,Z 231.979,A -85,B 0,C 180,E1 -8183.774,E2 -8183.774} C_VEL
LIN {X 0,Y 453.704,Z 231.968,A -85,B 0,C 180,E1 -8187.336,E2 -8187.336} C_VEL
LIN {X 0,Y 453.795,Z 231.958,A -85,B 0,C 180,E1 -8190,E2 -8190} C_VEL
LIN {X 0,Y 453.737,Z 231.963,A -85,B 0,C 180,E1 -8192.663,E2 -8192.663} C_VEL
LIN {X 0,Y 453.335,Z 232.191,A -85,B 0,C 180,E1 -8195.895,E2 -8195.895} C_VEL
LIN {X 0,Y 453.162,Z 238.742,A -85,B 0,C 180,E1 -8198.922,E2 -8198.922} C_VEL
LIN {X 0,Y 453.141,Z 246.423,A -85,B 0,C 180,E1 -8202.541,E2 -8202.541} C_VEL
LIN {X 0,Y 453.022,Z 253.488,A -85,B 0,C 180,E1 -8205.877,E2 -8205.877} C_VEL
LIN {X 0,Y 452.926,Z 260.083,A -85,B 0,C 180,E1 -8209.017,E2 -8209.017} C_VEL
LIN {X 0,Y 452.8,Z 267.086,A -85,B 0,C 180,E1 -8212.35,E2 -8212.35} C_VEL
LIN {X 0,Y 452.815,Z 271.779,A -85,B 0,C 180,E1 -8214.592,E2 -8214.592} C_VEL
LIN {X 0,Y 455.034,Z 284.932,A -85,B 0,C 180,E1 -8215.134,E2 -8215.134} C_VEL
LIN {X 0,Y 454.784,Z 294.52,A -85,B 0,C 180,E1 -8215.639,E2 -8215.639} C_VEL
LIN {X 0,Y 454.462,Z 303.363,A -85,B 0,C 180,E1 -8216.241,E2 -8216.241} C_VEL
LIN {X 0,Y 454.183,Z 311.258,A -85,B 0,C 180,E1 -8216.911,E2 -8216.911} C_VEL
LIN {X 0,Y 453.91,Z 318.651,A -85,B 0,C 180,E1 -8217.678,E2 -8217.678} C_VEL
LIN {X 0,Y 453.614,Z 325.342,A -85,B 0,C 180,E1 -8218.515,E2 -8218.515} C_VEL
LIN {X 0,Y 453.326,Z 331.714,A -85,B 0,C 180,E1 -8219.481,E2 -8219.481} C_VEL
LIN {X 0,Y 453.012,Z 338.573,A -85,B 0,C 180,E1 -8220.795,E2 -8220.795} C_VEL
LIN {X 0,Y 452.825,Z 342.819,A -85,B 0,C 180,E1 -8221.85,E2 -8221.85} C_VEL
LIN {X 0,Y 452.666,Z 346.47,A -85,B 0,C 180,E1 -8223.029,E2 -8223.029} C_VEL
LIN {X 0,Y 452.625,Z 348.714,A -85,B 0,C 180,E1 -8223.985,E2 -8223.985} C_VEL
LIN {X 0,Y 452.492,Z 350.497,A -85,B 0,C 180,E1 -8225.077,E2 -8225.077} C_VEL
LIN {X 0,Y 452.473,Z 351.509,A -85,B 0,C 180,E1 -8226.174,E2 -8226.174} C_VEL
LIN {X 0,Y 452.426,Z 351.657,A -85,B 0,C 180,E1 -8227.604,E2 -8227.604} C_VEL
LIN {X 0,Y 452.499,Z 350.561,A -85,B 0,C 180,E1 -8229.051,E2 -8229.051} C_VEL
LIN {X 0,Y 452.675,Z 347.599,A -85,B 0,C 180,E1 -8230.698,E2 -8230.698} C_VEL
LIN {X 0,Y 452.824,Z 344.348,A -85,B 0,C 180,E1 -8231.865,E2 -8231.865} C_VEL
LIN {X 0,Y 452.977,Z 341.2,A -85,B 0,C 180,E1 -8232.749,E2 -8232.749} C_VEL
LIN {X 0,Y 453.128,Z 337.121,A -85,B 0,C 180,E1 -8233.684,E2 -8233.684} C_VEL
LIN {X 0,Y 453.387,Z 331.694,A -85,B 0,C 180,E1 -8234.692,E2 -8234.692} C_VEL
LIN {X 0,Y 453.682,Z 325.526,A -85,B 0,C 180,E1 -8235.63,E2 -8235.63} C_VEL
LIN {X 0,Y 453.977,Z 319.112,A -85,B 0,C 180,E1 -8236.439,E2 -8236.439} C_VEL
LIN {X 0,Y 454.248,Z 311.702,A -85,B 0,C 180,E1 -8237.213,E2 -8237.213} C_VEL
LIN {X 0,Y 454.605,Z 303.543,A -85,B 0,C 180,E1 -8237.907,E2 -8237.907} C_VEL
LIN {X 0,Y 454.963,Z 292.903,A -85,B 0,C 180,E1 -8238.62,E2 -8238.62} C_VEL
LIN {X 0,Y 455.086,Z 284.614,A -85,B 0,C 180,E1 -8239.037,E2 -8239.037} C_VEL
LIN {X 0,Y 453.16,Z 273.876,A -85,B 0,C 180,E1 -8239.48,E2 -8239.48} C_VEL
LIN {X 0,Y 452.855,Z 272.271,A -85,B 0,C 180,E1 -8239.542,E2 -8239.542} C_VEL
LIN {X 0,Y 452.919,Z 265.496,A -85,B 0,C 180,E1 -8242.759,E2 -8242.759} C_VEL
LIN {X 0,Y 453.007,Z 258.54,A -85,B 0,C 180,E1 -8246.047,E2 -8246.047} C_VEL
LIN {X 0,Y 453.091,Z 251.788,A -85,B 0,C 180,E1 -8249.211,E2 -8249.211} C_VEL
LIN {X 0,Y 453.141,Z 245.283,A -85,B 0,C 180,E1 -8252.134,E2 -8252.134} C_VEL
LIN {X 0,Y 453.237,Z 237.242,A -85,B 0,C 180,E1 -8255.738,E2 -8255.738} C_VEL
LIN {X 0,Y 453.32,Z 232.026,A -85,B 0,C 180,E1 -8258.036,E2 -8258.036} C_VEL
LIN {X 0,Y 453.525,Z 231.995,A -85,B 0,C 180,E1 -8261.009,E2 -8261.009} C_VEL
LIN {X 0,Y 453.572,Z 231.988,A -85,B 0,C 180,E1 -8263.88,E2 -8263.88} C_VEL
LIN {X 0,Y 453.566,Z 231.989,A -85,B 0,C 180,E1 -8267.471,E2 -8267.471} C_VEL
LIN {X 0,Y 453.595,Z 231.984,A -85,B 0,C 180,E1 -8271.087,E2 -8271.087} C_VEL
LIN {X 0,Y 453.649,Z 231.978,A -85,B 0,C 180,E1 -8273.774,E2 -8273.774} C_VEL
LIN {X 0,Y 453.747,Z 231.966,A -85,B 0,C 180,E1 -8277.337,E2 -8277.337} C_VEL
LIN {X 0,Y 453.826,Z 231.956,A -85,B 0,C 180,E1 -8280,E2 -8280} C_VEL
LIN {X 0,Y 453.747,Z 231.967,A -85,B 0,C 180,E1 -8282.663,E2 -8282.663} C_VEL
LIN {X 0,Y 453.654,Z 231.978,A -85,B 0,C 180,E1 -8286.226,E2 -8286.226} C_VEL
LIN {X 0,Y 453.594,Z 231.984,A -85,B 0,C 180,E1 -8288.913,E2 -8288.913} C_VEL
LIN {X 0,Y 453.566,Z 231.988,A -85,B 0,C 180,E1 -8292.529,E2 -8292.529} C_VEL
LIN {X 0,Y 453.547,Z 231.988,A -85,B 0,C 180,E1 -8296.196,E2 -8296.196} C_VEL
LIN {X 0,Y 453.52,Z 231.993,A -85,B 0,C 180,E1 -8299.04,E2 -8299.04} C_VEL
LIN {X 0,Y 453.479,Z 231.999,A -85,B 0,C 180,E1 -8301.836,E2 -8301.836} C_VEL
LIN {X 0,Y 453.498,Z 231.996,A -85,B 0,C 180,E1 -8304.735,E2 -8304.735} C_VEL
LIN {X 0,Y 453.531,Z 231.992,A -85,B 0,C 180,E1 -8307.959,E2 -8307.959} C_VEL
LIN {X 0,Y 453.467,Z 231.999,A -85,B 0,C 180,E1 -8311.525,E2 -8311.525} C_VEL
LIN {X 0,Y 453.484,Z 231.998,A -85,B 0,C 180,E1 -8314.776,E2 -8314.776} C_VEL
LIN {X 0,Y 453.466,Z 232.002,A -85,B 0,C 180,E1 -8318.312,E2 -8318.312} C_VEL
LIN {X 0,Y 453.496,Z 231.999,A -85,B 0,C 180,E1 -8320.609,E2 -8320.609} C_VEL
LIN {X 0,Y 453.456,Z 232.002,A -85,B 0,C 180,E1 -8323.244,E2 -8323.244} C_VEL
LIN {X 0,Y 453.465,Z 232.002,A -85,B 0,C 180,E1 -8325.779,E2 -8325.779} C_VEL
LIN {X 0,Y 453.525,Z 232.007,A -85,B 0,C 180,E1 -8329.102,E2 -8329.102} C_VEL
LIN {X 0,Y 454.804,Z 239.417,A -85,B 0,C 180,E1 -8332.5,E2 -8332.5} C_VEL
LIN {X 0,Y 455.222,Z 243.007,A -85,B 0,C 180,E1 -8334.079,E2 -8334.079} C_VEL
LIN {X 0,Y 455.007,Z 248.146,A -85,B 0,C 180,E1 -8336.217,E2 -8336.217} C_VEL
LIN {X 0,Y 454.489,Z 255.842,A -85,B 0,C 180,E1 -8339.316,E2 -8339.316} C_VEL
LIN {X 0,Y 454.03,Z 263.542,A -85,B 0,C 180,E1 -8342.33,E2 -8342.33} C_VEL
LIN {X 0,Y 453.639,Z 272.451,A -85,B 0,C 180,E1 -8345.732,E2 -8345.732} C_VEL
LIN {X 0,Y 453.257,Z 281.542,A -85,B 0,C 180,E1 -8349.107,E2 -8349.107} C_VEL
LIN {X 0,Y 452.958,Z 290.549,A -85,B 0,C 180,E1 -8352.389,E2 -8352.389} C_VEL
LIN {X 0,Y 452.861,Z 295.614,A -85,B 0,C 180,E1 -8354.216,E2 -8354.216} C_VEL
LIN {X 0,Y 454.836,Z 310.183,A -85,B 0,C 180,E1 -8354.72,E2 -8354.72} C_VEL
LIN {X 0,Y 455.809,Z 319.456,A -85,B 0,C 180,E1 -8355.147,E2 -8355.147} C_VEL
LIN {X 0,Y 455.246,Z 331.658,A -85,B 0,C 180,E1 -8355.814,E2 -8355.814} C_VEL
LIN {X 0,Y 454.656,Z 343.823,A -85,B 0,C 180,E1 -8356.683,E2 -8356.683} C_VEL
LIN {X 0,Y 454.106,Z 355.236,A -85,B 0,C 180,E1 -8357.713,E2 -8357.713} C_VEL
LIN {X 0,Y 453.634,Z 365.162,A -85,B 0,C 180,E1 -8358.834,E2 -8358.834} C_VEL
LIN {X 0,Y 453.181,Z 374.823,A -85,B 0,C 180,E1 -8360.178,E2 -8360.178} C_VEL
LIN {X 0,Y 452.872,Z 382.519,A -85,B 0,C 180,E1 -8361.522,E2 -8361.522} C_VEL
LIN {X 0,Y 452.69,Z 388.707,A -85,B 0,C 180,E1 -8362.866,E2 -8362.866} C_VEL
LIN {X 0,Y 452.568,Z 393.604,A -85,B 0,C 180,E1 -8364.207,E2 -8364.207} C_VEL
LIN {X 0,Y 452.497,Z 397.347,A -85,B 0,C 180,E1 -8365.546,E2 -8365.546} C_VEL
LIN {X 0,Y 452.525,Z 399.273,A -85,B 0,C 180,E1 -8366.438,E2 -8366.438} C_VEL
LIN {X 0,Y 452.543,Z 400.74,A -85,B 0,C 180,E1 -8367.33,E2 -8367.33} C_VEL
LIN {X 0,Y 452.538,Z 401.755,A -85,B 0,C 180,E1 -8368.22,E2 -8368.22} C_VEL
LIN {X 0,Y 452.492,Z 402.365,A -85,B 0,C 180,E1 -8369.11,E2 -8369.11} C_VEL
LIN {X 0,Y 452.471,Z 402.574,A -85,B 0,C 180,E1 -8370,E2 -8370} C_VEL
LIN {X 0,Y 452.492,Z 402.343,A -85,B 0,C 180,E1 -8370.89,E2 -8370.89} C_VEL
LIN {X 0,Y 452.523,Z 401.687,A -85,B 0,C 180,E1 -8371.78,E2 -8371.78} C_VEL
LIN {X 0,Y 452.544,Z 400.625,A -85,B 0,C 180,E1 -8372.671,E2 -8372.671} C_VEL
LIN {X 0,Y 452.527,Z 399.148,A -85,B 0,C 180,E1 -8373.562,E2 -8373.562} C_VEL
LIN {X 0,Y 452.557,Z 396.062,A -85,B 0,C 180,E1 -8374.9,E2 -8374.9} C_VEL
LIN {X 0,Y 452.611,Z 391.335,A -85,B 0,C 180,E1 -8376.396,E2 -8376.396} C_VEL
LIN {X 0,Y 452.775,Z 385.523,A -85,B 0,C 180,E1 -8377.806,E2 -8377.806} C_VEL
LIN {X 0,Y 453.006,Z 378.582,A -85,B 0,C 180,E1 -8379.15,E2 -8379.15} C_VEL
LIN {X 0,Y 453.36,Z 370.031,A -85,B 0,C 180,E1 -8380.495,E2 -8380.495} C_VEL
LIN {X 0,Y 453.84,Z 361.283,A -85,B 0,C 180,E1 -8381.614,E2 -8381.614} C_VEL
LIN {X 0,Y 454.287,Z 350.243,A -85,B 0,C 180,E1 -8382.77,E2 -8382.77} C_VEL
LIN {X 0,Y 454.927,Z 338.728,A -85,B 0,C 180,E1 -8383.741,E2 -8383.741} C_VEL
LIN {X 0,Y 455.587,Z 327.032,A -85,B 0,C 180,E1 -8384.518,E2 -8384.518} C_VEL
LIN {X 0,Y 455.811,Z 317.731,A -85,B 0,C 180,E1 -8385.024,E2 -8385.024} C_VEL
LIN {X 0,Y 454.39,Z 303.157,A -85,B 0,C 180,E1 -8385.69,E2 -8385.69} C_VEL
LIN {X 0,Y 452.771,Z 293.273,A -85,B 0,C 180,E1 -8386.069,E2 -8386.069} C_VEL
LIN {X 0,Y 452.991,Z 284.99,A -85,B 0,C 180,E1 -8389.015,E2 -8389.015} C_VEL
LIN {X 0,Y 453.291,Z 276.001,A -85,B 0,C 180,E1 -8392.325,E2 -8392.325} C_VEL
LIN {X 0,Y 453.679,Z 266.474,A -85,B 0,C 180,E1 -8396.04,E2 -8396.04} C_VEL
LIN {X 0,Y 454.133,Z 259.024,A -85,B 0,C 180,E1 -8399.176,E2 -8399.176} C_VEL
LIN {X 0,Y 454.661,Z 253.349,A -85,B 0,C 180,E1 -8401.769,E2 -8401.769} C_VEL
LIN {X 0,Y 455.174,Z 249.35,A -85,B 0,C 180,E1 -8403.77,E2 -8403.77} C_VEL
LIN {X 0,Y 455.446,Z 245.565,A -85,B 0,C 180,E1 -8405.901,E2 -8405.901} C_VEL
LIN {X 0,Y 455.26,Z 242.221,A -85,B 0,C 180,E1 -8408.134,E2 -8408.134} C_VEL
LIN {X 0,Y 454.772,Z 239.11,A -85,B 0,C 180,E1 -8410.778,E2 -8410.778} C_VEL
LIN {X 0,Y 454.36,Z 236.911,A -85,B 0,C 180,E1 -8413.365,E2 -8413.365} C_VEL
LIN {X 0,Y 454.101,Z 235.551,A -85,B 0,C 180,E1 -8415.857,E2 -8415.857} C_VEL
LIN {X 0,Y 453.986,Z 234.902,A -85,B 0,C 180,E1 -8418.266,E2 -8418.266} C_VEL
LIN {X 0,Y 453.962,Z 234.838,A -85,B 0,C 180,E1 -8420.722,E2 -8420.722} C_VEL
LIN {X 0,Y 454.042,Z 235.53,A -85,B 0,C 180,E1 -8423.971,E2 -8423.971} C_VEL
LIN {X 0,Y 453.859,Z 236.912,A -85,B 0,C 180,E1 -8427.182,E2 -8427.182} C_VEL
LIN {X 0,Y 453.595,Z 238.736,A -85,B 0,C 180,E1 -8430.277,E2 -8430.277} C_VEL
LIN {X 0,Y 453.416,Z 240.794,A -85,B 0,C 180,E1 -8433.288,E2 -8433.288} C_VEL
LIN {X 0,Y 453.25,Z 243.04,A -85,B 0,C 180,E1 -8436.225,E2 -8436.225} C_VEL
LIN {X 0,Y 453.074,Z 245.417,A -85,B 0,C 180,E1 -8439.098,E2 -8439.098} C_VEL
LIN {X 0,Y 453.005,Z 247.882,A -85,B 0,C 180,E1 -8441.924,E2 -8441.924} C_VEL
LIN {X 0,Y 452.953,Z 250.793,A -85,B 0,C 180,E1 -8445.095,E2 -8445.095} C_VEL
LIN {X 0,Y 456.419,Z 264.025,A -85,B 0,C 180,E1 -8445.737,E2 -8445.737} C_VEL
LIN {X 0,Y 456.793,Z 268.072,A -85,B 0,C 180,E1 -8445.939,E2 -8445.939} C_VEL
LIN {X 0,Y 456.24,Z 280.983,A -85,B 0,C 180,E1 -8446.64,E2 -8446.64} C_VEL
LIN {X 0,Y 455.632,Z 293.38,A -85,B 0,C 180,E1 -8447.529,E2 -8447.529} C_VEL
LIN {X 0,Y 455.071,Z 304.425,A -85,B 0,C 180,E1 -8448.531,E2 -8448.531} C_VEL
LIN {X 0,Y 454.604,Z 313.43,A -85,B 0,C 180,E1 -8449.534,E2 -8449.534} C_VEL
LIN {X 0,Y 454.023,Z 323.15,A -85,B 0,C 180,E1 -8450.871,E2 -8450.871} C_VEL
LIN {X 0,Y 453.566,Z 331.12,A -85,B 0,C 180,E1 -8452.23,E2 -8452.23} C_VEL
LIN {X 0,Y 453.233,Z 336.877,A -85,B 0,C 180,E1 -8453.449,E2 -8453.449} C_VEL
LIN {X 0,Y 453.128,Z 341.494,A -85,B 0,C 180,E1 -8454.66,E2 -8454.66} C_VEL
LIN {X 0,Y 452.953,Z 345.523,A -85,B 0,C 180,E1 -8455.996,E2 -8455.996} C_VEL
LIN {X 0,Y 452.759,Z 348.502,A -85,B 0,C 180,E1 -8457.331,E2 -8457.331} C_VEL
LIN {X 0,Y 452.591,Z 349.962,A -85,B 0,C 180,E1 -8458.22,E2 -8458.22} C_VEL
LIN {X 0,Y 452.481,Z 351.568,A -85,B 0,C 180,E1 -8460,E2 -8460} C_VEL
LIN {X 0,Y 452.498,Z 351.782,A -85,B 0,C 180,E1 -8460.89,E2 -8460.89} C_VEL
LIN {X 0,Y 452.578,Z 351.579,A -85,B 0,C 180,E1 -8461.78,E2 -8461.78} C_VEL
LIN {X 0,Y 452.674,Z 349.925,A -85,B 0,C 180,E1 -8463.561,E2 -8463.561} C_VEL
LIN {X 0,Y 452.629,Z 348.507,A -85,B 0,C 180,E1 -8464.453,E2 -8464.453} C_VEL
LIN {X 0,Y 452.797,Z 345.519,A -85,B 0,C 180,E1 -8465.79,E2 -8465.79} C_VEL
LIN {X 0,Y 452.86,Z 341.486,A -85,B 0,C 180,E1 -8467.132,E2 -8467.132} C_VEL
LIN {X 0,Y 453.166,Z 335.264,A -85,B 0,C 180,E1 -8468.697,E2 -8468.697} C_VEL
LIN {X 0,Y 453.459,Z 328.469,A -85,B 0,C 180,E1 -8470.042,E2 -8470.042} C_VEL
LIN {X 0,Y 453.898,Z 320.043,A -85,B 0,C 180,E1 -8471.386,E2 -8471.386} C_VEL
LIN {X 0,Y 454.355,Z 310.047,A -85,B 0,C 180,E1 -8472.66,E2 -8472.66} C_VEL
LIN {X 0,Y 454.858,Z 299.552,A -85,B 0,C 180,E1 -8473.743,E2 -8473.743} C_VEL
LIN {X 0,Y 455.429,Z 288.719,A -85,B 0,C 180,E1 -8474.637,E2 -8474.637} C_VEL
LIN {X 0,Y 455.895,Z 277.117,A -85,B 0,C 180,E1 -8475.4,E2 -8475.4} C_VEL
LIN {X 0,Y 456.246,Z 265.129,A -85,B 0,C 180,E1 -8476.011,E2 -8476.011} C_VEL
LIN {X 0,Y 453.521,Z 252.421,A -85,B 0,C 180,E1 -8476.571,E2 -8476.571} C_VEL
LIN {X 0,Y 452.609,Z 248.125,A -85,B 0,C 180,E1 -8476.746,E2 -8476.746} C_VEL
LIN {X 0,Y 452.645,Z 245.552,A -85,B 0,C 180,E1 -8479.03,E2 -8479.03} C_VEL
LIN {X 0,Y 452.661,Z 242.393,A -85,B 0,C 180,E1 -8481.878,E2 -8481.878} C_VEL
LIN {X 0,Y 452.802,Z 238.161,A -85,B 0,C 180,E1 -8485.76,E2 -8485.76} C_VEL
LIN {X 0,Y 452.787,Z 234.958,A -85,B 0,C 180,E1 -8488.762,E2 -8488.762} C_VEL
LIN {X 0,Y 452.831,Z 232.201,A -85,B 0,C 180,E1 -8491.393,E2 -8491.393} C_VEL
LIN {X 0,Y 453.157,Z 232.04,A -85,B 0,C 180,E1 -8493.94,E2 -8493.94} C_VEL
LIN {X 0,Y 453.392,Z 232.009,A -85,B 0,C 180,E1 -8496.288,E2 -8496.288} C_VEL
LIN {X 0,Y 453.467,Z 232,A -85,B 0,C 180,E1 -8499.453,E2 -8499.453} C_VEL
LIN {X 0,Y 453.463,Z 232,A -85,B 0,C 180,E1 -8501.932,E2 -8501.932} C_VEL
LIN {X 0,Y 453.485,Z 231.998,A -85,B 0,C 180,E1 -8505.471,E2 -8505.471} C_VEL
LIN {X 0,Y 453.456,Z 231.999,A -85,B 0,C 180,E1 -8508.206,E2 -8508.206} C_VEL
LIN {X 0,Y 453.441,Z 232.004,A -85,B 0,C 180,E1 -8510.802,E2 -8510.802} C_VEL
LIN {X 0,Y 453.444,Z 231.998,A -85,B 0,C 180,E1 -8513.916,E2 -8513.916} C_VEL
LIN {X 0,Y 453.478,Z 231.996,A -85,B 0,C 180,E1 -8517.15,E2 -8517.15} C_VEL
LIN {X 0,Y 453.471,Z 232.001,A -85,B 0,C 180,E1 -8520.268,E2 -8520.268} C_VEL
LIN {X 0,Y 453.476,Z 231.998,A -85,B 0,C 180,E1 -8523.292,E2 -8523.292} C_VEL
LIN {X 0,Y 453.501,Z 231.996,A -85,B 0,C 180,E1 -8526.238,E2 -8526.238} C_VEL
LIN {X 0,Y 453.487,Z 231.997,A -85,B 0,C 180,E1 -8529.118,E2 -8529.118} C_VEL
LIN {X 0,Y 453.507,Z 231.994,A -85,B 0,C 180,E1 -8531.944,E2 -8531.944} C_VEL
LIN {X 0,Y 453.542,Z 231.992,A -85,B 0,C 180,E1 -8534.726,E2 -8534.726} C_VEL
LIN {X 0,Y 453.556,Z 231.987,A -85,B 0,C 180,E1 -8537.681,E2 -8537.681} C_VEL
LIN {X 0,Y 452.873,Z 232.076,A -85,B 0,C 180,E1 -8538.422,E2 -8538.422} C_VEL
LIN {X 0,Y 450.01,Z 232.429,A -85,B 0,C 180,E1 -8539.626,E2 -8539.626} C_VEL
LIN {X 0,Y 447.608,Z 232.729,A -85,B 0,C 180,E1 -8540.597,E2 -8540.597} C_VEL
LIN {X 0,Y 446.592,Z 232.854,A -85,B 0,C 180,E1 -8541.348,E2 -8541.348} C_VEL
LIN {X 0,Y 446.518,Z 232.863,A -85,B 0,C 180,E1 -8541.602,E2 -8541.602} C_VEL
LIN {X 0,Y 446.619,Z 232.851,A -85,B 0,C 180,E1 -8544.582,E2 -8544.582} C_VEL
LIN {X 0,Y 446.66,Z 232.846,A -85,B 0,C 180,E1 -8548.196,E2 -8548.196} C_VEL
LIN {X 0,Y 446.765,Z 232.834,A -85,B 0,C 180,E1 -8550,E2 -8550} C_VEL
LIN {X 0,Y 446.683,Z 232.842,A -85,B 0,C 180,E1 -8552.705,E2 -8552.705} C_VEL
LIN {X 0,Y 446.297,Z 233.084,A -85,B 0,C 180,E1 -8555.875,E2 -8555.875} C_VEL
LIN {X 0,Y 446.099,Z 239.935,A -85,B 0,C 180,E1 -8559.064,E2 -8559.064} C_VEL
LIN {X 0,Y 446.107,Z 246.92,A -85,B 0,C 180,E1 -8562.377,E2 -8562.377} C_VEL
LIN {X 0,Y 445.965,Z 254.525,A -85,B 0,C 180,E1 -8565.99,E2 -8565.99} C_VEL
LIN {X 0,Y 445.825,Z 261.514,A -85,B 0,C 180,E1 -8569.332,E2 -8569.332} C_VEL
LIN {X 0,Y 445.739,Z 268.596,A -85,B 0,C 180,E1 -8572.724,E2 -8572.724} C_VEL
LIN {X 0,Y 445.768,Z 272.13,A -85,B 0,C 180,E1 -8574.416,E2 -8574.416} C_VEL
LIN {X 0,Y 447.835,Z 283.755,A -85,B 0,C 180,E1 -8574.884,E2 -8574.884} C_VEL
LIN {X 0,Y 447.941,Z 289.844,A -85,B 0,C 180,E1 -8575.187,E2 -8575.187} C_VEL
LIN {X 0,Y 447.638,Z 300.435,A -85,B 0,C 180,E1 -8575.829,E2 -8575.829} C_VEL
LIN {X 0,Y 447.286,Z 310.202,A -85,B 0,C 180,E1 -8576.626,E2 -8576.626} C_VEL
LIN {X 0,Y 446.973,Z 317.641,A -85,B 0,C 180,E1 -8577.382,E2 -8577.382} C_VEL
LIN {X 0,Y 446.651,Z 324.454,A -85,B 0,C 180,E1 -8578.218,E2 -8578.218} C_VEL
LIN {X 0,Y 446.421,Z 329.535,A -85,B 0,C 180,E1 -8578.953,E2 -8578.953} C_VEL
LIN {X 0,Y 446.14,Z 335.287,A -85,B 0,C 180,E1 -8579.955,E2 -8579.955} C_VEL
LIN {X 0,Y 445.917,Z 340.472,A -85,B 0,C 180,E1 -8581.075,E2 -8581.075} C_VEL
LIN {X 0,Y 445.733,Z 343.912,A -85,B 0,C 180,E1 -8581.995,E2 -8581.995} C_VEL
LIN {X 0,Y 445.595,Z 348.177,A -85,B 0,C 180,E1 -8583.506,E2 -8583.506} C_VEL
LIN {X 0,Y 445.434,Z 350.676,A -85,B 0,C 180,E1 -8584.87,E2 -8584.87} C_VEL
LIN {X 0,Y 445.363,Z 351.981,A -85,B 0,C 180,E1 -8586.409,E2 -8586.409} C_VEL
LIN {X 0,Y 445.355,Z 351.925,A -85,B 0,C 180,E1 -8587.984,E2 -8587.984} C_VEL
LIN {X 0,Y 445.452,Z 350.623,A -85,B 0,C 180,E1 -8589.368,E2 -8589.368} C_VEL
LIN {X 0,Y 445.615,Z 347.904,A -85,B 0,C 180,E1 -8590.796,E2 -8590.796} C_VEL
LIN {X 0,Y 445.753,Z 345.125,A -85,B 0,C 180,E1 -8591.828,E2 -8591.828} C_VEL
LIN {X 0,Y 446.001,Z 340.539,A -85,B 0,C 180,E1 -8593.103,E2 -8593.103} C_VEL
LIN {X 0,Y 446.168,Z 335.829,A -85,B 0,C 180,E1 -8594.133,E2 -8594.133} C_VEL
LIN {X 0,Y 446.444,Z 330.371,A -85,B 0,C 180,E1 -8595.105,E2 -8595.105} C_VEL
LIN {X 0,Y 446.825,Z 322.787,A -85,B 0,C 180,E1 -8596.206,E2 -8596.206} C_VEL
LIN {X 0,Y 447.225,Z 313.514,A -85,B 0,C 180,E1 -8597.244,E2 -8597.244} C_VEL
LIN {X 0,Y 447.581,Z 306.308,A -85,B 0,C 180,E1 -8597.896,E2 -8597.896} C_VEL
LIN {X 0,Y 447.854,Z 297.675,A -85,B 0,C 180,E1 -8598.532,E2 -8598.532} C_VEL
LIN {X 0,Y 448.151,Z 288.49,A -85,B 0,C 180,E1 -8599.059,E2 -8599.059} C_VEL
LIN {X 0,Y 447.923,Z 283.975,A -85,B 0,C 180,E1 -8599.284,E2 -8599.284} C_VEL
LIN {X 0,Y 445.996,Z 273.735,A -85,B 0,C 180,E1 -8599.708,E2 -8599.708} C_VEL
LIN {X 0,Y 445.834,Z 272.603,A -85,B 0,C 180,E1 -8599.764,E2 -8599.764} C_VEL
LIN {X 0,Y 445.888,Z 265.365,A -85,B 0,C 180,E1 -8603.205,E2 -8603.205} C_VEL
LIN {X 0,Y 446.002,Z 258.114,A -85,B 0,C 180,E1 -8606.633,E2 -8606.633} C_VEL
LIN {X 0,Y 446.071,Z 251.55,A -85,B 0,C 180,E1 -8609.723,E2 -8609.723} C_VEL
LIN {X 0,Y 446.11,Z 244.746,A -85,B 0,C 180,E1 -8612.815,E2 -8612.815} C_VEL
LIN {X 0,Y 446.201,Z 237.612,A -85,B 0,C 180,E1 -8616,E2 -8616} C_VEL
LIN {X 0,Y 446.278,Z 232.904,A -85,B 0,C 180,E1 -8618.096,E2 -8618.096} C_VEL
LIN {X 0,Y 446.475,Z 232.873,A -85,B 0,C 180,E1 -8620.816,E2 -8620.816} C_VEL
LIN {X 0,Y 446.51,Z 232.869,A -85,B 0,C 180,E1 -8624.48,E2 -8624.48} C_VEL
LIN {X 0,Y 446.521,Z 232.869,A -85,B 0,C 180,E1 -8628.193,E2 -8628.193} C_VEL
LIN {X 0,Y 446.541,Z 232.864,A -85,B 0,C 180,E1 -8630.945,E2 -8630.945} C_VEL
LIN {X 0,Y 446.618,Z 232.854,A -85,B 0,C 180,E1 -8633.676,E2 -8633.676} C_VEL
LIN {X 0,Y 446.694,Z 232.844,A -85,B 0,C 180,E1 -8637.295,E2 -8637.295} C_VEL
LIN {X 0,Y 446.796,Z 232.832,A -85,B 0,C 180,E1 -8640,E2 -8640} C_VEL
LIN {X 0,Y 446.693,Z 232.845,A -85,B 0,C 180,E1 -8642.705,E2 -8642.705} C_VEL
LIN {X 0,Y 446.622,Z 232.853,A -85,B 0,C 180,E1 -8646.324,E2 -8646.324} C_VEL
LIN {X 0,Y 446.539,Z 232.863,A -85,B 0,C 180,E1 -8649.055,E2 -8649.055} C_VEL
LIN {X 0,Y 446.524,Z 232.865,A -85,B 0,C 180,E1 -8652.73,E2 -8652.73} C_VEL
LIN {X 0,Y 446.498,Z 232.866,A -85,B 0,C 180,E1 -8656.227,E2 -8656.227} C_VEL
LIN {X 0,Y 446.471,Z 232.873,A -85,B 0,C 180,E1 -8659.303,E2 -8659.303} C_VEL
LIN {X 0,Y 446.42,Z 232.878,A -85,B 0,C 180,E1 -8662.199,E2 -8662.199} C_VEL
LIN {X 0,Y 446.441,Z 232.878,A -85,B 0,C 180,E1 -8665.153,E2 -8665.153} C_VEL
LIN {X 0,Y 446.487,Z 232.87,A -85,B 0,C 180,E1 -8668.179,E2 -8668.179} C_VEL
LIN {X 0,Y 446.42,Z 232.877,A -85,B 0,C 180,E1 -8671.775,E2 -8671.775} C_VEL
LIN {X 0,Y 446.425,Z 232.877,A -85,B 0,C 180,E1 -8674.523,E2 -8674.523} C_VEL
LIN {X 0,Y 446.417,Z 232.879,A -85,B 0,C 180,E1 -8678.079,E2 -8678.079} C_VEL
LIN {X 0,Y 446.428,Z 232.877,A -85,B 0,C 180,E1 -8680.918,E2 -8680.918} C_VEL
LIN {X 0,Y 446.402,Z 232.881,A -85,B 0,C 180,E1 -8683.846,E2 -8683.846} C_VEL
LIN {X 0,Y 446.4,Z 232.883,A -85,B 0,C 180,E1 -8686.403,E2 -8686.403} C_VEL
LIN {X 0,Y 446.468,Z 232.948,A -85,B 0,C 180,E1 -8688.881,E2 -8688.881} C_VEL
LIN {X 0,Y 447.721,Z 240.147,A -85,B 0,C 180,E1 -8692.252,E2 -8692.252} C_VEL
LIN {X 0,Y 448.22,Z 244.028,A -85,B 0,C 180,E1 -8693.985,E2 -8693.985} C_VEL
LIN {X 0,Y 447.976,Z 249.367,A -85,B 0,C 180,E1 -8696.252,E2 -8696.252} C_VEL
LIN {X 0,Y 447.537,Z 255.544,A -85,B 0,C 180,E1 -8698.787,E2 -8698.787} C_VEL
LIN {X 0,Y 447.065,Z 263.241,A -85,B 0,C 180,E1 -8701.861,E2 -8701.861} C_VEL
LIN {X 0,Y 446.635,Z 272.206,A -85,B 0,C 180,E1 -8705.355,E2 -8705.355} C_VEL
LIN {X 0,Y 446.192,Z 281.195,A -85,B 0,C 180,E1 -8708.76,E2 -8708.76} C_VEL
LIN {X 0,Y 445.936,Z 288.876,A -85,B 0,C 180,E1 -8711.627,E2 -8711.627} C_VEL
LIN {X 0,Y 445.81,Z 295.48,A -85,B 0,C 180,E1 -8714.006,E2 -8714.006} C_VEL
LIN {X 0,Y 447.759,Z 309.618,A -85,B 0,C 180,E1 -8714.499,E2 -8714.499} C_VEL
LIN {X 0,Y 448.818,Z 320.746,A -85,B 0,C 180,E1 -8715.027,E2 -8715.027} C_VEL
LIN {X 0,Y 448.225,Z 332.488,A -85,B 0,C 180,E1 -8715.703,E2 -8715.703} C_VEL
LIN {X 0,Y 447.649,Z 343.949,A -85,B 0,C 180,E1 -8716.547,E2 -8716.547} C_VEL
LIN {X 0,Y 447.125,Z 354.525,A -85,B 0,C 180,E1 -8717.519,E2 -8717.519} C_VEL
LIN {X 0,Y 446.625,Z 364.508,A -85,B 0,C 180,E1 -8718.656,E2 -8718.656} C_VEL
LIN {X 0,Y 446.112,Z 374.218,A -85,B 0,C 180,E1 -8720.021,E2 -8720.021} C_VEL
LIN {X 0,Y 445.813,Z 381.97,A -85,B 0,C 180,E1 -8721.387,E2 -8721.387} C_VEL
LIN {X 0,Y 445.613,Z 388.192,A -85,B 0,C 180,E1 -8722.752,E2 -8722.752} C_VEL
LIN {X 0,Y 445.489,Z 392.543,A -85,B 0,C 180,E1 -8723.934,E2 -8723.934} C_VEL
LIN {X 0,Y 445.422,Z 396.886,A -85,B 0,C 180,E1 -8725.475,E2 -8725.475} C_VEL
LIN {X 0,Y 445.427,Z 398.821,A -85,B 0,C 180,E1 -8726.382,E2 -8726.382} C_VEL
LIN {X 0,Y 445.467,Z 400.309,A -85,B 0,C 180,E1 -8727.287,E2 -8727.287} C_VEL
LIN {X 0,Y 445.45,Z 401.332,A -85,B 0,C 180,E1 -8728.192,E2 -8728.192} C_VEL
LIN {X 0,Y 445.429,Z 401.95,A -85,B 0,C 180,E1 -8729.096,E2 -8729.096} C_VEL
LIN {X 0,Y 445.406,Z 402.165,A -85,B 0,C 180,E1 -8730,E2 -8730} C_VEL
LIN {X 0,Y 445.429,Z 401.948,A -85,B 0,C 180,E1 -8730.904,E2 -8730.904} C_VEL
LIN {X 0,Y 445.437,Z 401.295,A -85,B 0,C 180,E1 -8731.808,E2 -8731.808} C_VEL
LIN {X 0,Y 445.467,Z 400.238,A -85,B 0,C 180,E1 -8732.713,E2 -8732.713} C_VEL
LIN {X 0,Y 445.426,Z 398.764,A -85,B 0,C 180,E1 -8733.619,E2 -8733.619} C_VEL
LIN {X 0,Y 445.487,Z 395.682,A -85,B 0,C 180,E1 -8734.978,E2 -8734.978} C_VEL
LIN {X 0,Y 445.529,Z 391.375,A -85,B 0,C 180,E1 -8736.386,E2 -8736.386} C_VEL
LIN {X 0,Y 445.711,Z 385.173,A -85,B 0,C 180,E1 -8737.931,E2 -8737.931} C_VEL
LIN {X 0,Y 445.949,Z 378.254,A -85,B 0,C 180,E1 -8739.296,E2 -8739.296} C_VEL
LIN {X 0,Y 446.326,Z 369.725,A -85,B 0,C 180,E1 -8740.662,E2 -8740.662} C_VEL
LIN {X 0,Y 446.851,Z 361.036,A -85,B 0,C 180,E1 -8741.798,E2 -8741.798} C_VEL
LIN {X 0,Y 447.294,Z 350.917,A -85,B 0,C 180,E1 -8742.89,E2 -8742.89} C_VEL
LIN {X 0,Y 447.949,Z 340.081,A -85,B 0,C 180,E1 -8743.843,E2 -8743.843} C_VEL
LIN {X 0,Y 448.615,Z 329.007,A -85,B 0,C 180,E1 -8744.632,E2 -8744.632} C_VEL
LIN {X 0,Y 449.019,Z 319.164,A -85,B 0,C 180,E1 -8745.199,E2 -8745.199} C_VEL
LIN {X 0,Y 447.781,Z 305.831,A -85,B 0,C 180,E1 -8745.859,E2 -8745.859} C_VEL
LIN {X 0,Y 445.707,Z 292.737,A -85,B 0,C 180,E1 -8746.4,E2 -8746.4} C_VEL
LIN {X 0,Y 445.949,Z 284.706,A -85,B 0,C 180,E1 -8749.327,E2 -8749.327} C_VEL
LIN {X 0,Y 446.265,Z 275.796,A -85,B 0,C 180,E1 -8752.696,E2 -8752.696} C_VEL
LIN {X 0,Y 446.67,Z 266.924,A -85,B 0,C 180,E1 -8756.253,E2 -8756.253} C_VEL
LIN {X 0,Y 447.12,Z 260.184,A -85,B 0,C 180,E1 -8759.162,E2 -8759.162} C_VEL
LIN {X 0,Y 447.789,Z 253.651,A -85,B 0,C 180,E1 -8762.251,E2 -8762.251} C_VEL
LIN {X 0,Y 448.314,Z 249.63,A -85,B 0,C 180,E1 -8764.358,E2 -8764.358} C_VEL
LIN {X 0,Y 448.496,Z 245.989,A -85,B 0,C 180,E1 -8766.546,E2 -8766.546} C_VEL
LIN {X 0,Y 448.182,Z 242.828,A -85,B 0,C 180,E1 -8768.848,E2 -8768.848} C_VEL
LIN {X 0,Y 447.775,Z 240.217,A -85,B 0,C 180,E1 -8771.24,E2 -8771.24} C_VEL
LIN {X 0,Y 447.4,Z 238.231,A -85,B 0,C 180,E1 -8773.731,E2 -8773.731} C_VEL
LIN {X 0,Y 447.126,Z 236.934,A -85,B 0,C 180,E1 -8776.306,E2 -8776.306} C_VEL
LIN {X 0,Y 447.025,Z 236.321,A -85,B 0,C 180,E1 -8778.995,E2 -8778.995} C_VEL
LIN {X 0,Y 447.02,Z 236.465,A -85,B 0,C 180,E1 -8782.182,E2 -8782.182} C_VEL
LIN {X 0,Y 447.025,Z 237.166,A -85,B 0,C 180,E1 -8784.839,E2 -8784.839} C_VEL
LIN {X 0,Y 446.801,Z 238.421,A -85,B 0,C 180,E1 -8787.669,E2 -8787.669} C_VEL
LIN {X 0,Y 446.529,Z 240.232,A -85,B 0,C 180,E1 -8790.796,E2 -8790.796} C_VEL
LIN {X 0,Y 446.358,Z 242.28,A -85,B 0,C 180,E1 -8793.841,E2 -8793.841} C_VEL
LIN {X 0,Y 446.154,Z 244.527,A -85,B 0,C 180,E1 -8796.808,E2 -8796.808} C_VEL
LIN {X 0,Y 445.988,Z 246.897,A -85,B 0,C 180,E1 -8799.715,E2 -8799.715} C_VEL
LIN {X 0,Y 445.942,Z 249.367,A -85,B 0,C 180,E1 -8802.576,E2 -8802.576} C_VEL
LIN {X 0,Y 445.951,Z 251.508,A -85,B 0,C 180,E1 -8804.782,E2 -8804.782} C_VEL
LIN {X 0,Y 449.531,Z 264.734,A -85,B 0,C 180,E1 -8805.456,E2 -8805.456} C_VEL
LIN {X 0,Y 450.081,Z 268.167,A -85,B 0,C 180,E1 -8805.643,E2 -8805.643} C_VEL
LIN {X 0,Y 449.497,Z 280.786,A -85,B 0,C 180,E1 -8806.336,E2 -8806.336} C_VEL
LIN {X 0,Y 449.006,Z 291.747,A -85,B 0,C 180,E1 -8807.112,E2 -8807.112} C_VEL
LIN {X 0,Y 448.295,Z 303.138,A -85,B 0,C 180,E1 -8808.126,E2 -8808.126} C_VEL
LIN {X 0,Y 447.771,Z 312.399,A -85,B 0,C 180,E1 -8809.144,E2 -8809.144} C_VEL
LIN {X 0,Y 447.302,Z 320.921,A -85,B 0,C 180,E1 -8810.276,E2 -8810.276} C_VEL
LIN {X 0,Y 446.793,Z 328.002,A -85,B 0,C 180,E1 -8811.406,E2 -8811.406} C_VEL
LIN {X 0,Y 446.363,Z 334.969,A -85,B 0,C 180,E1 -8812.764,E2 -8812.764} C_VEL
LIN {X 0,Y 446.098,Z 340.506,A -85,B 0,C 180,E1 -8814.122,E2 -8814.122} C_VEL
LIN {X 0,Y 445.895,Z 344.863,A -85,B 0,C 180,E1 -8815.48,E2 -8815.48} C_VEL
LIN {X 0,Y 445.906,Z 347.144,A -85,B 0,C 180,E1 -8816.385,E2 -8816.385} C_VEL
LIN {X 0,Y 445.711,Z 349.013,A -85,B 0,C 180,E1 -8817.289,E2 -8817.289} C_VEL
LIN {X 0,Y 445.535,Z 350.44,A -85,B 0,C 180,E1 -8818.192,E2 -8818.192} C_VEL
LIN {X 0,Y 445.416,Z 352.004,A -85,B 0,C 180,E1 -8820,E2 -8820} C_VEL
LIN {X 0,Y 445.436,Z 352.198,A -85,B 0,C 180,E1 -8820.904,E2 -8820.904} C_VEL
LIN {X 0,Y 445.49,Z 351.96,A -85,B 0,C 180,E1 -8821.808,E2 -8821.808} C_VEL
LIN {X 0,Y 445.538,Z 351.306,A -85,B 0,C 180,E1 -8822.713,E2 -8822.713} C_VEL
LIN {X 0,Y 445.608,Z 350.259,A -85,B 0,C 180,E1 -8823.617,E2 -8823.617} C_VEL
LIN {X 0,Y 445.544,Z 348.814,A -85,B 0,C 180,E1 -8824.524,E2 -8824.524} C_VEL
LIN {X 0,Y 445.742,Z 345.779,A -85,B 0,C 180,E1 -8825.882,E2 -8825.882} C_VEL
LIN {X 0,Y 445.792,Z 341.691,A -85,B 0,C 180,E1 -8827.246,E2 -8827.246} C_VEL
LIN {X 0,Y 446.14,Z 335.388,A -85,B 0,C 180,E1 -8828.835,E2 -8828.835} C_VEL
LIN {X 0,Y 446.454,Z 328.526,A -85,B 0,C 180,E1 -8830.201,E2 -8830.201} C_VEL
LIN {X 0,Y 446.92,Z 319.997,A -85,B 0,C 180,E1 -8831.566,E2 -8831.566} C_VEL
LIN {X 0,Y 447.358,Z 311.227,A -85,B 0,C 180,E1 -8832.706,E2 -8832.706} C_VEL
LIN {X 0,Y 447.858,Z 300.48,A -85,B 0,C 180,E1 -8833.846,E2 -8833.846} C_VEL
LIN {X 0,Y 448.445,Z 289.838,A -85,B 0,C 180,E1 -8834.754,E2 -8834.754} C_VEL
LIN {X 0,Y 448.942,Z 278.42,A -85,B 0,C 180,E1 -8835.53,E2 -8835.53} C_VEL
LIN {X 0,Y 449.327,Z 265.98,A -85,B 0,C 180,E1 -8836.184,E2 -8836.184} C_VEL
LIN {X 0,Y 446.478,Z 253.056,A -85,B 0,C 180,E1 -8836.777,E2 -8836.777} C_VEL
LIN {X 0,Y 445.538,Z 248.453,A -85,B 0,C 180,E1 -8836.967,E2 -8836.967} C_VEL
LIN {X 0,Y 445.574,Z 245.79,A -85,B 0,C 180,E1 -8839.344,E2 -8839.344} C_VEL
LIN {X 0,Y 445.566,Z 242.604,A -85,B 0,C 180,E1 -8842.245,E2 -8842.245} C_VEL
LIN {X 0,Y 445.664,Z 239.395,A -85,B 0,C 180,E1 -8845.2,E2 -8845.2} C_VEL
LIN {X 0,Y 445.717,Z 236.165,A -85,B 0,C 180,E1 -8848.232,E2 -8848.232} C_VEL
LIN {X 0,Y 445.767,Z 232.962,A -85,B 0,C 180,E1 -8851.351,E2 -8851.351} C_VEL
LIN {X 0,Y 446.176,Z 232.909,A -85,B 0,C 180,E1 -8854.546,E2 -8854.546} C_VEL
LIN {X 0,Y 446.352,Z 232.887,A -85,B 0,C 180,E1 -8856.75,E2 -8856.75} C_VEL
LIN {X 0,Y 446.436,Z 232.876,A -85,B 0,C 180,E1 -8859.521,E2 -8859.521} C_VEL
LIN {X 0,Y 446.421,Z 232.876,A -85,B 0,C 180,E1 -8862.606,E2 -8862.606} C_VEL
LIN {X 0,Y 446.454,Z 232.874,A -85,B 0,C 180,E1 -8865.104,E2 -8865.104} C_VEL
LIN {X 0,Y 446.409,Z 232.877,A -85,B 0,C 180,E1 -8868.606,E2 -8868.606} C_VEL
LIN {X 0,Y 446.399,Z 232.876,A -85,B 0,C 180,E1 -8871.924,E2 -8871.924} C_VEL
LIN {X 0,Y 446.423,Z 232.874,A -85,B 0,C 180,E1 -8875.476,E2 -8875.476} C_VEL
LIN {X 0,Y 446.418,Z 232.878,A -85,B 0,C 180,E1 -8878.699,E2 -8878.699} C_VEL
LIN {X 0,Y 446.454,Z 232.872,A -85,B 0,C 180,E1 -8881.83,E2 -8881.83} C_VEL
LIN {X 0,Y 446.447,Z 232.873,A -85,B 0,C 180,E1 -8884.847,E2 -8884.847} C_VEL
LIN {X 0,Y 446.453,Z 232.873,A -85,B 0,C 180,E1 -8888.245,E2 -8888.245} C_VEL
LIN {X 0,Y 446.456,Z 232.874,A -85,B 0,C 180,E1 -8891.649,E2 -8891.649} C_VEL
LIN {X 0,Y 446.511,Z 232.867,A -85,B 0,C 180,E1 -8894.48,E2 -8894.48} C_VEL
LIN {X 0,Y 446.521,Z 232.866,A -85,B 0,C 180,E1 -8898.193,E2 -8898.193} C_VEL
LIN {X 0,Y 446.518,Z 232.863,A -85,B 0,C 180,E1 -8901.602,E2 -8901.602} C_VEL
LIN {X 0,Y 445.87,Z 232.948,A -85,B 0,C 180,E1 -8902.355,E2 -8902.355} C_VEL
LIN {X 0,Y 443.009,Z 233.305,A -85,B 0,C 180,E1 -8903.579,E2 -8903.579} C_VEL
LIN {X 0,Y 440.56,Z 233.608,A -85,B 0,C 180,E1 -8904.566,E2 -8904.566} C_VEL
LIN {X 0,Y 439.487,Z 233.739,A -85,B 0,C 180,E1 -8905.329,E2 -8905.329} C_VEL
LIN {X 0,Y 439.389,Z 233.75,A -85,B 0,C 180,E1 -8905.588,E2 -8905.588} C_VEL
LIN {X 0,Y 439.629,Z 233.722,A -85,B 0,C 180,E1 -8908.168,E2 -8908.168} C_VEL
LIN {X 0,Y 439.714,Z 233.712,A -85,B 0,C 180,E1 -8910,E2 -8910} C_VEL
LIN {X 0,Y 439.631,Z 233.72,A -85,B 0,C 180,E1 -8912.749,E2 -8912.749} C_VEL
LIN {X 0,Y 439.261,Z 233.966,A -85,B 0,C 180,E1 -8915.854,E2 -8915.854} C_VEL
LIN {X 0,Y 439.095,Z 239.149,A -85,B 0,C 180,E1 -8918.282,E2 -8918.282} C_VEL
LIN {X 0,Y 439.047,Z 246.996,A -85,B 0,C 180,E1 -8922.011,E2 -8922.011} C_VEL
LIN {X 0,Y 438.92,Z 252.94,A -85,B 0,C 180,E1 -8924.844,E2 -8924.844} C_VEL
LIN {X 0,Y 438.834,Z 258.928,A -85,B 0,C 180,E1 -8927.715,E2 -8927.715} C_VEL
LIN {X 0,Y 438.723,Z 266.021,A -85,B 0,C 180,E1 -8931.127,E2 -8931.127} C_VEL
LIN {X 0,Y 438.708,Z 272.445,A -85,B 0,C 180,E1 -8934.22,E2 -8934.22} C_VEL
LIN {X 0,Y 440.921,Z 284.838,A -85,B 0,C 180,E1 -8934.734,E2 -8934.734} C_VEL
LIN {X 0,Y 440.881,Z 295.312,A -85,B 0,C 180,E1 -8935.304,E2 -8935.304} C_VEL
LIN {X 0,Y 440.56,Z 303.76,A -85,B 0,C 180,E1 -8935.893,E2 -8935.893} C_VEL
LIN {X 0,Y 440.213,Z 312.021,A -85,B 0,C 180,E1 -8936.614,E2 -8936.614} C_VEL
LIN {X 0,Y 439.881,Z 320.009,A -85,B 0,C 180,E1 -8937.473,E2 -8937.473} C_VEL
LIN {X 0,Y 439.531,Z 327.235,A -85,B 0,C 180,E1 -8938.425,E2 -8938.425} C_VEL
LIN {X 0,Y 439.13,Z 335.12,A -85,B 0,C 180,E1 -8939.745,E2 -8939.745} C_VEL
LIN {X 0,Y 438.898,Z 340.171,A -85,B 0,C 180,E1 -8940.825,E2 -8940.825} C_VEL
LIN {X 0,Y 438.673,Z 344.264,A -85,B 0,C 180,E1 -8941.917,E2 -8941.917} C_VEL
LIN {X 0,Y 438.515,Z 347.472,A -85,B 0,C 180,E1 -8943.019,E2 -8943.019} C_VEL
LIN {X 0,Y 438.446,Z 349.858,A -85,B 0,C 180,E1 -8944.127,E2 -8944.127} C_VEL
LIN {X 0,Y 438.314,Z 351.494,A -85,B 0,C 180,E1 -8945.256,E2 -8945.256} C_VEL
LIN {X 0,Y 438.282,Z 352.471,A -85,B 0,C 180,E1 -8946.7,E2 -8946.7} C_VEL
LIN {X 0,Y 438.273,Z 352.229,A -85,B 0,C 180,E1 -8948.21,E2 -8948.21} C_VEL
LIN {X 0,Y 438.405,Z 350.229,A -85,B 0,C 180,E1 -8949.884,E2 -8949.884} C_VEL
LIN {X 0,Y 438.597,Z 347.637,A -85,B 0,C 180,E1 -8951.138,E2 -8951.138} C_VEL
LIN {X 0,Y 438.739,Z 344.347,A -85,B 0,C 180,E1 -8952.282,E2 -8952.282} C_VEL
LIN {X 0,Y 438.975,Z 339.749,A -85,B 0,C 180,E1 -8953.506,E2 -8953.506} C_VEL
LIN {X 0,Y 439.287,Z 333.726,A -85,B 0,C 180,E1 -8954.744,E2 -8954.744} C_VEL
LIN {X 0,Y 439.629,Z 327.217,A -85,B 0,C 180,E1 -8955.795,E2 -8955.795} C_VEL
LIN {X 0,Y 440.008,Z 320.408,A -85,B 0,C 180,E1 -8956.696,E2 -8956.696} C_VEL
LIN {X 0,Y 440.391,Z 312.076,A -85,B 0,C 180,E1 -8957.595,E2 -8957.595} C_VEL
LIN {X 0,Y 440.804,Z 302.2,A -85,B 0,C 180,E1 -8958.443,E2 -8958.443} C_VEL
LIN {X 0,Y 441.197,Z 291.319,A -85,B 0,C 180,E1 -8959.131,E2 -8959.131} C_VEL
LIN {X 0,Y 441.103,Z 285.476,A -85,B 0,C 180,E1 -8959.439,E2 -8959.439} C_VEL
LIN {X 0,Y 438.993,Z 274.304,A -85,B 0,C 180,E1 -8959.918,E2 -8959.918} C_VEL
LIN {X 0,Y 438.789,Z 272.985,A -85,B 0,C 180,E1 -8959.971,E2 -8959.971} C_VEL
LIN {X 0,Y 438.842,Z 266.223,A -85,B 0,C 180,E1 -8963.201,E2 -8963.201} C_VEL
LIN {X 0,Y 438.926,Z 259.565,A -85,B 0,C 180,E1 -8966.368,E2 -8966.368} C_VEL
LIN {X 0,Y 438.995,Z 253.563,A -85,B 0,C 180,E1 -8969.183,E2 -8969.183} C_VEL
LIN {X 0,Y 439.094,Z 248.269,A -85,B 0,C 180,E1 -8971.68,E2 -8971.68} C_VEL
LIN {X 0,Y 439.19,Z 239.917,A -85,B 0,C 180,E1 -8975.414,E2 -8975.414} C_VEL
LIN {X 0,Y 439.253,Z 233.778,A -85,B 0,C 180,E1 -8978.236,E2 -8978.236} C_VEL
LIN {X 0,Y 439.427,Z 233.751,A -85,B 0,C 180,E1 -8981.345,E2 -8981.345} C_VEL
LIN {X 0,Y 439.465,Z 233.745,A -85,B 0,C 180,E1 -8984.224,E2 -8984.224} C_VEL
LIN {X 0,Y 439.487,Z 233.744,A -85,B 0,C 180,E1 -8988.001,E2 -8988.001} C_VEL
LIN {X 0,Y 439.536,Z 233.738,A -85,B 0,C 180,E1 -8991.726,E2 -8991.726} C_VEL
LIN {X 0,Y 439.61,Z 233.727,A -85,B 0,C 180,E1 -8994.496,E2 -8994.496} C_VEL
LIN {X 0,Y 439.637,Z 233.724,A -85,B 0,C 180,E1 -8998.168,E2 -8998.168} C_VEL
LIN {X 0,Y 439.766,Z 233.708,A -85,B 0,C 180,E1 -9000,E2 -9000} C_VEL
LIN {X 0,Y 439.643,Z 233.723,A -85,B 0,C 180,E1 -9002.749,E2 -9002.749} C_VEL
LIN {X 0,Y 439.594,Z 233.728,A -85,B 0,C 180,E1 -9006.425,E2 -9006.425} C_VEL
LIN {X 0,Y 439.501,Z 233.74,A -85,B 0,C 180,E1 -9009.202,E2 -9009.202} C_VEL
LIN {X 0,Y 439.468,Z 233.745,A -85,B 0,C 180,E1 -9012.937,E2 -9012.937} C_VEL
LIN {X 0,Y 439.449,Z 233.744,A -85,B 0,C 180,E1 -9016.348,E2 -9016.348} C_VEL
LIN {X 0,Y 439.404,Z 233.752,A -85,B 0,C 180,E1 -9019.626,E2 -9019.626} C_VEL
LIN {X 0,Y 439.365,Z 233.758,A -85,B 0,C 180,E1 -9022.575,E2 -9022.575} C_VEL
LIN {X 0,Y 439.389,Z 233.754,A -85,B 0,C 180,E1 -9025.586,E2 -9025.586} C_VEL
LIN {X 0,Y 439.419,Z 233.751,A -85,B 0,C 180,E1 -9028.673,E2 -9028.673} C_VEL
LIN {X 0,Y 439.37,Z 233.756,A -85,B 0,C 180,E1 -9032.03,E2 -9032.03} C_VEL
LIN {X 0,Y 439.394,Z 233.752,A -85,B 0,C 180,E1 -9035.34,E2 -9035.34} C_VEL
LIN {X 0,Y 439.385,Z 233.754,A -85,B 0,C 180,E1 -9038.595,E2 -9038.595} C_VEL
LIN {X 0,Y 439.39,Z 233.754,A -85,B 0,C 180,E1 -9041.257,E2 -9041.257} C_VEL
LIN {X 0,Y 439.401,Z 233.753,A -85,B 0,C 180,E1 -9044.729,E2 -9044.729} C_VEL
LIN {X 0,Y 439.433,Z 233.802,A -85,B 0,C 180,E1 -9048.628,E2 -9048.628} C_VEL
LIN {X 0,Y 440.476,Z 239.842,A -85,B 0,C 180,E1 -9051.518,E2 -9051.518} C_VEL
LIN {X 0,Y 441.218,Z 245.008,A -85,B 0,C 180,E1 -9053.888,E2 -9053.888} C_VEL
LIN {X 0,Y 440.999,Z 250.139,A -85,B 0,C 180,E1 -9056.098,E2 -9056.098} C_VEL
LIN {X 0,Y 440.519,Z 256.532,A -85,B 0,C 180,E1 -9058.768,E2 -9058.768} C_VEL
LIN {X 0,Y 440,Z 264.293,A -85,B 0,C 180,E1 -9061.924,E2 -9061.924} C_VEL
LIN {X 0,Y 439.615,Z 271.874,A -85,B 0,C 180,E1 -9064.935,E2 -9064.935} C_VEL
LIN {X 0,Y 439.16,Z 280.823,A -85,B 0,C 180,E1 -9068.403,E2 -9068.403} C_VEL
LIN {X 0,Y 438.875,Z 288.48,A -85,B 0,C 180,E1 -9071.321,E2 -9071.321} C_VEL
LIN {X 0,Y 438.755,Z 294.971,A -85,B 0,C 180,E1 -9073.76,E2 -9073.76} C_VEL
LIN {X 0,Y 440.803,Z 310.363,A -85,B 0,C 180,E1 -9074.333,E2 -9074.333} C_VEL
LIN {X 0,Y 441.857,Z 320.732,A -85,B 0,C 180,E1 -9074.844,E2 -9074.844} C_VEL
LIN {X 0,Y 441.204,Z 333.227,A -85,B 0,C 180,E1 -9075.588,E2 -9075.588} C_VEL
LIN {X 0,Y 440.594,Z 344.866,A -85,B 0,C 180,E1 -9076.479,E2 -9076.479} C_VEL
LIN {X 0,Y 440.019,Z 355.895,A -85,B 0,C 180,E1 -9077.548,E2 -9077.548} C_VEL
LIN {X 0,Y 439.515,Z 365.586,A -85,B 0,C 180,E1 -9078.704,E2 -9078.704} C_VEL
LIN {X 0,Y 439.058,Z 373.561,A -85,B 0,C 180,E1 -9079.859,E2 -9079.859} C_VEL
LIN {X 0,Y 438.742,Z 381.382,A -85,B 0,C 180,E1 -9081.247,E2 -9081.247} C_VEL
LIN {X 0,Y 438.536,Z 387.643,A -85,B 0,C 180,E1 -9082.634,E2 -9082.634} C_VEL
LIN {X 0,Y 438.391,Z 392.456,A -85,B 0,C 180,E1 -9083.972,E2 -9083.972} C_VEL
LIN {X 0,Y 438.351,Z 396.406,A -85,B 0,C 180,E1 -9085.402,E2 -9085.402} C_VEL
LIN {X 0,Y 438.331,Z 398.353,A -85,B 0,C 180,E1 -9086.323,E2 -9086.323} C_VEL
LIN {X 0,Y 438.392,Z 399.866,A -85,B 0,C 180,E1 -9087.243,E2 -9087.243} C_VEL
LIN {X 0,Y 438.366,Z 400.902,A -85,B 0,C 180,E1 -9088.163,E2 -9088.163} C_VEL
LIN {X 0,Y 438.368,Z 401.531,A -85,B 0,C 180,E1 -9089.082,E2 -9089.082} C_VEL
LIN {X 0,Y 438.344,Z 401.754,A -85,B 0,C 180,E1 -9090,E2 -9090} C_VEL
LIN {X 0,Y 438.351,Z 401.553,A -85,B 0,C 180,E1 -9090.919,E2 -9090.919} C_VEL
LIN {X 0,Y 438.354,Z 400.905,A -85,B 0,C 180,E1 -9091.838,E2 -9091.838} C_VEL
LIN {X 0,Y 438.392,Z 399.855,A -85,B 0,C 180,E1 -9092.757,E2 -9092.757} C_VEL
LIN {X 0,Y 438.327,Z 398.385,A -85,B 0,C 180,E1 -9093.677,E2 -9093.677} C_VEL
LIN {X 0,Y 438.417,Z 395.318,A -85,B 0,C 180,E1 -9095.058,E2 -9095.058} C_VEL
LIN {X 0,Y 438.448,Z 391.176,A -85,B 0,C 180,E1 -9096.443,E2 -9096.443} C_VEL
LIN {X 0,Y 438.657,Z 384.849,A -85,B 0,C 180,E1 -9098.059,E2 -9098.059} C_VEL
LIN {X 0,Y 438.906,Z 377.961,A -85,B 0,C 180,E1 -9099.447,E2 -9099.447} C_VEL
LIN {X 0,Y 439.315,Z 369.466,A -85,B 0,C 180,E1 -9100.835,E2 -9100.835} C_VEL
LIN {X 0,Y 439.868,Z 360.844,A -85,B 0,C 180,E1 -9101.988,E2 -9101.988} C_VEL
LIN {X 0,Y 440.376,Z 350.411,A -85,B 0,C 180,E1 -9103.137,E2 -9103.137} C_VEL
LIN {X 0,Y 441.131,Z 338.694,A -85,B 0,C 180,E1 -9104.179,E2 -9104.179} C_VEL
LIN {X 0,Y 441.88,Z 327.404,A -85,B 0,C 180,E1 -9104.979,E2 -9104.979} C_VEL
LIN {X 0,Y 442.109,Z 319.566,A -85,B 0,C 180,E1 -9105.443,E2 -9105.443} C_VEL
LIN {X 0,Y 441.103,Z 307.515,A -85,B 0,C 180,E1 -9106.076,E2 -9106.076} C_VEL
LIN {X 0,Y 439.154,Z 295.003,A -85,B 0,C 180,E1 -9106.617,E2 -9106.617} C_VEL
LIN {X 0,Y 438.638,Z 292.247,A -85,B 0,C 180,E1 -9106.738,E2 -9106.738} C_VEL
LIN {X 0,Y 438.892,Z 284.449,A -85,B 0,C 180,E1 -9109.65,E2 -9109.65} C_VEL
LIN {X 0,Y 439.202,Z 276.873,A -85,B 0,C 180,E1 -9112.585,E2 -9112.585} C_VEL
LIN {X 0,Y 439.601,Z 268.455,A -85,B 0,C 180,E1 -9116.022,E2 -9116.022} C_VEL
LIN {X 0,Y 440.1,Z 261.363,A -85,B 0,C 180,E1 -9119.148,E2 -9119.148} C_VEL
LIN {X 0,Y 440.808,Z 254.797,A -85,B 0,C 180,E1 -9122.327,E2 -9122.327} C_VEL
LIN {X 0,Y 441.279,Z 251.493,A -85,B 0,C 180,E1 -9124.088,E2 -9124.088} C_VEL
LIN {X 0,Y 441.513,Z 248.149,A -85,B 0,C 180,E1 -9126.084,E2 -9126.084} C_VEL
LIN {X 0,Y 441.356,Z 244.904,A -85,B 0,C 180,E1 -9128.391,E2 -9128.391} C_VEL
LIN {X 0,Y 440.8,Z 241.58,A -85,B 0,C 180,E1 -9131.465,E2 -9131.465} C_VEL
LIN {X 0,Y 440.379,Z 239.272,A -85,B 0,C 180,E1 -9134.604,E2 -9134.604} C_VEL
LIN {X 0,Y 440.124,Z 238.016,A -85,B 0,C 180,E1 -9137.881,E2 -9137.881} C_VEL
LIN {X 0,Y 440.079,Z 237.746,A -85,B 0,C 180,E1 -9140.298,E2 -9140.298} C_VEL
LIN {X 0,Y 440.069,Z 238.199,A -85,B 0,C 180,E1 -9143.779,E2 -9143.779} C_VEL
LIN {X 0,Y 439.951,Z 239.004,A -85,B 0,C 180,E1 -9146.169,E2 -9146.169} C_VEL
LIN {X 0,Y 439.658,Z 240.496,A -85,B 0,C 180,E1 -9149.234,E2 -9149.234} C_VEL
LIN {X 0,Y 439.438,Z 242.382,A -85,B 0,C 180,E1 -9152.367,E2 -9152.367} C_VEL
LIN {X 0,Y 439.206,Z 244.784,A -85,B 0,C 180,E1 -9155.797,E2 -9155.797} C_VEL
LIN {X 0,Y 438.988,Z 247.585,A -85,B 0,C 180,E1 -9159.377,E2 -9159.377} C_VEL
LIN {X 0,Y 438.921,Z 250.029,A -85,B 0,C 180,E1 -9162.288,E2 -9162.288} C_VEL
LIN {X 0,Y 438.902,Z 251.898,A -85,B 0,C 180,E1 -9164.412,E2 -9164.412} C_VEL
LIN {X 0,Y 442.982,Z 266.805,A -85,B 0,C 180,E1 -9165.236,E2 -9165.236} C_VEL
LIN {X 0,Y 443.343,Z 270.133,A -85,B 0,C 180,E1 -9165.424,E2 -9165.424} C_VEL
LIN {X 0,Y 442.723,Z 282.206,A -85,B 0,C 180,E1 -9166.115,E2 -9166.115} C_VEL
LIN {X 0,Y 442.041,Z 294.345,A -85,B 0,C 180,E1 -9167.022,E2 -9167.022} C_VEL
LIN {X 0,Y 441.343,Z 305.303,A -85,B 0,C 180,E1 -9168.053,E2 -9168.053} C_VEL
LIN {X 0,Y 440.774,Z 315.154,A -85,B 0,C 180,E1 -9169.202,E2 -9169.202} C_VEL
LIN {X 0,Y 440.123,Z 324.697,A -85,B 0,C 180,E1 -9170.58,E2 -9170.58} C_VEL
LIN {X 0,Y 439.594,Z 332.394,A -85,B 0,C 180,E1 -9171.959,E2 -9171.959} C_VEL
LIN {X 0,Y 439.06,Z 339.434,A -85,B 0,C 180,E1 -9173.567,E2 -9173.567} C_VEL
LIN {X 0,Y 438.956,Z 344.115,A -85,B 0,C 180,E1 -9174.948,E2 -9174.948} C_VEL
LIN {X 0,Y 438.865,Z 347.69,A -85,B 0,C 180,E1 -9176.327,E2 -9176.327} C_VEL
LIN {X 0,Y 438.665,Z 349.537,A -85,B 0,C 180,E1 -9177.245,E2 -9177.245} C_VEL
LIN {X 0,Y 438.481,Z 350.924,A -85,B 0,C 180,E1 -9178.163,E2 -9178.163} C_VEL
LIN {X 0,Y 438.353,Z 352.446,A -85,B 0,C 180,E1 -9180,E2 -9180} C_VEL
LIN {X 0,Y 438.375,Z 352.614,A -85,B 0,C 180,E1 -9180.919,E2 -9180.919} C_VEL
LIN {X 0,Y 438.405,Z 352.339,A -85,B 0,C 180,E1 -9181.837,E2 -9181.837} C_VEL
LIN {X 0,Y 438.466,Z 351.661,A -85,B 0,C 180,E1 -9182.756,E2 -9182.756} C_VEL
LIN {X 0,Y 438.523,Z 350.588,A -85,B 0,C 180,E1 -9183.676,E2 -9183.676} C_VEL
LIN {X 0,Y 438.464,Z 349.103,A -85,B 0,C 180,E1 -9184.597,E2 -9184.597} C_VEL
LIN {X 0,Y 438.666,Z 346.02,A -85,B 0,C 180,E1 -9185.978,E2 -9185.978} C_VEL
LIN {X 0,Y 438.75,Z 341.871,A -85,B 0,C 180,E1 -9187.363,E2 -9187.363} C_VEL
LIN {X 0,Y 439.092,Z 335.493,A -85,B 0,C 180,E1 -9188.978,E2 -9188.978} C_VEL
LIN {X 0,Y 439.436,Z 328.561,A -85,B 0,C 180,E1 -9190.365,E2 -9190.365} C_VEL
LIN {X 0,Y 439.83,Z 321.496,A -85,B 0,C 180,E1 -9191.522,E2 -9191.522} C_VEL
LIN {X 0,Y 440.331,Z 313.002,A -85,B 0,C 180,E1 -9192.677,E2 -9192.677} C_VEL
LIN {X 0,Y 440.747,Z 303.962,A -85,B 0,C 180,E1 -9193.696,E2 -9193.696} C_VEL
LIN {X 0,Y 441.351,Z 292.277,A -85,B 0,C 180,E1 -9194.761,E2 -9194.761} C_VEL
LIN {X 0,Y 441.955,Z 281.187,A -85,B 0,C 180,E1 -9195.566,E2 -9195.566} C_VEL
LIN {X 0,Y 442.38,Z 268.447,A -85,B 0,C 180,E1 -9196.283,E2 -9196.283} C_VEL
LIN {X 0,Y 441.684,Z 263.735,A -85,B 0,C 180,E1 -9196.525,E2 -9196.525} C_VEL
LIN {X 0,Y 438.617,Z 249.811,A -85,B 0,C 180,E1 -9197.126,E2 -9197.126} C_VEL
LIN {X 0,Y 438.478,Z 248.785,A -85,B 0,C 180,E1 -9197.188,E2 -9197.188} C_VEL
LIN {X 0,Y 438.496,Z 246.023,A -85,B 0,C 180,E1 -9199.669,E2 -9199.669} C_VEL
LIN {X 0,Y 438.488,Z 242.8,A -85,B 0,C 180,E1 -9202.623,E2 -9202.623} C_VEL
LIN {X 0,Y 438.666,Z 238.941,A -85,B 0,C 180,E1 -9206.207,E2 -9206.207} C_VEL
LIN {X 0,Y 438.694,Z 235.188,A -85,B 0,C 180,E1 -9209.777,E2 -9209.777} C_VEL
LIN {X 0,Y 438.673,Z 234.096,A -85,B 0,C 180,E1 -9210.842,E2 -9210.842} C_VEL
LIN {X 0,Y 438.944,Z 233.811,A -85,B 0,C 180,E1 -9212.983,E2 -9212.983} C_VEL
LIN {X 0,Y 439.209,Z 233.779,A -85,B 0,C 180,E1 -9215.305,E2 -9215.305} C_VEL
LIN {X 0,Y 439.368,Z 233.757,A -85,B 0,C 180,E1 -9218.597,E2 -9218.597} C_VEL
LIN {X 0,Y 439.385,Z 233.754,A -85,B 0,C 180,E1 -9221.256,E2 -9221.256} C_VEL
LIN {X 0,Y 439.402,Z 233.75,A -85,B 0,C 180,E1 -9224.73,E2 -9224.73} C_VEL
LIN {X 0,Y 439.361,Z 233.755,A -85,B 0,C 180,E1 -9227.791,E2 -9227.791} C_VEL
LIN {X 0,Y 439.357,Z 233.755,A -85,B 0,C 180,E1 -9231.402,E2 -9231.402} C_VEL
LIN {X 0,Y 439.394,Z 233.754,A -85,B 0,C 180,E1 -9234.843,E2 -9234.843} C_VEL
LIN {X 0,Y 439.373,Z 233.754,A -85,B 0,C 180,E1 -9238.139,E2 -9238.139} C_VEL
LIN {X 0,Y 439.413,Z 233.749,A -85,B 0,C 180,E1 -9241.604,E2 -9241.604} C_VEL
LIN {X 0,Y 439.384,Z 233.754,A -85,B 0,C 180,E1 -9244.414,E2 -9244.414} C_VEL
LIN {X 0,Y 439.368,Z 233.755,A -85,B 0,C 180,E1 -9247.424,E2 -9247.424} C_VEL
LIN {X 0,Y 439.445,Z 233.746,A -85,B 0,C 180,E1 -9250.663,E2 -9250.663} C_VEL
LIN {X 0,Y 439.466,Z 233.743,A -85,B 0,C 180,E1 -9254.224,E2 -9254.224} C_VEL
LIN {X 0,Y 439.487,Z 233.741,A -85,B 0,C 180,E1 -9258.001,E2 -9258.001} C_VEL
LIN {X 0,Y 439.505,Z 233.738,A -85,B 0,C 180,E1 -9261.725,E2 -9261.725} C_VEL
LIN {X 0,Y 439.594,Z 233.726,A -85,B 0,C 180,E1 -9264.495,E2 -9264.495} C_VEL
LIN {X 0,Y 439.389,Z 233.75,A -85,B 0,C 180,E1 -9265.588,E2 -9265.588} C_VEL
